//     PlcTask Outputs/GVL_iXlinker.EtherCAT_Master_BKCUCX.TcTerminals210_EK1100_1.TcTerminals210_1BK1250.A_0361_KL_3361_1005_1_Ch_Oscilloscope.Channel_1.Data_Out_8 <-> Channel 1/Data Out 8
//     PlcTask Outputs/GVL_iXlinker.EtherCAT_Master_BKCUCX.TcTerminals210_EK1100_1.TcTerminals210_1BK1250.A_0361_KL_3361_1005_1_Ch_Oscilloscope.Channel_1.Data_Out_9 <-> Channel 1/Data Out 9
//     PlcTask Outputs/GVL_iXlinker.EtherCAT_Master_BKCUCX.TcTerminals210_EK1100_1.TcTerminals210_1BK1250.A_0361_KL_3361_1005_1_Ch_Oscilloscope.Channel_1.Data_Out_10 <-> Channel 1/Data Out 10
//   PLC/PLC Instance <-> EtherCAT Master BKCUCX/TcTerminals210_EK1100_1/TcTerminals210_1BK1250/A_0362(KL 3362, 2 Ch. Oscilloscope)
//     PlcTask Inputs/GVL_iXlinker.EtherCAT_Master_BKCUCX.TcTerminals210_EK1100_1.TcTerminals210_1BK1250.A_0362_KL_3362_2_Ch_Oscilloscope.Channel_1.State <-> Channel 1/State
//     PlcTask Inputs/GVL_iXlinker.EtherCAT_Master_BKCUCX.TcTerminals210_EK1100_1.TcTerminals210_1BK1250.A_0362_KL_3362_2_Ch_Oscilloscope.Channel_2.State <-> Channel 2/State
//     PlcTask Inputs/GVL_iXlinker.EtherCAT_Master_BKCUCX.TcTerminals210_EK1100_1.TcTerminals210_1BK1250.A_0362_KL_3362_2_Ch_Oscilloscope.Channel_1.Data_In <-> Channel 1/Data In
//     PlcTask Inputs/GVL_iXlinker.EtherCAT_Master_BKCUCX.TcTerminals210_EK1100_1.TcTerminals210_1BK1250.A_0362_KL_3362_2_Ch_Oscilloscope.Channel_2.Data_In <-> Channel 2/Data In
//     PlcTask Outputs/GVL_iXlinker.EtherCAT_Master_BKCUCX.TcTerminals210_EK1100_1.TcTerminals210_1BK1250.A_0362_KL_3362_2_Ch_Oscilloscope.Channel_1.Ctrl <-> Channel 1/Ctrl
//     PlcTask Outputs/GVL_iXlinker.EtherCAT_Master_BKCUCX.TcTerminals210_EK1100_1.TcTerminals210_1BK1250.A_0362_KL_3362_2_Ch_Oscilloscope.Channel_2.Ctrl <-> Channel 2/Ctrl
//     PlcTask Outputs/GVL_iXlinker.EtherCAT_Master_BKCUCX.TcTerminals210_EK1100_1.TcTerminals210_1BK1250.A_0362_KL_3362_2_Ch_Oscilloscope.Channel_1.Data_Out <-> Channel 1/Data Out
//     PlcTask Outputs/GVL_iXlinker.EtherCAT_Master_BKCUCX.TcTerminals210_EK1100_1.TcTerminals210_1BK1250.A_0362_KL_3362_2_Ch_Oscilloscope.Channel_2.Data_Out <-> Channel 2/Data Out
//   PLC/PLC Instance <-> EtherCAT Master BKCUCX/TcTerminals210_EK1100_2
//     PlcTask Inputs/GVL_iXlinker.EtherCAT_Master_BKCUCX.TcTerminals210_EK1100_2.InfoData.State <-> InfoData/State
//   PLC/PLC Instance <-> EtherCAT Master BKCUCX/TcTerminals210_EK1100_2/TcTerminals210_2BK1250
//     PlcTask Inputs/GVL_iXlinker.EtherCAT_Master_BKCUCX.TcTerminals210_EK1100_2.TcTerminals210_2BK1250.Inputs.CouplerState <-> Inputs/CouplerState
//     PlcTask Inputs/GVL_iXlinker.EtherCAT_Master_BKCUCX.TcTerminals210_EK1100_2.TcTerminals210_2BK1250.Outputs.CouplerCtrl <-> Outputs/CouplerCtrl
//     PlcTask Inputs/GVL_iXlinker.EtherCAT_Master_BKCUCX.TcTerminals210_EK1100_2.TcTerminals210_2BK1250.WcState.WcState <-> WcState/WcState
//     PlcTask Inputs/GVL_iXlinker.EtherCAT_Master_BKCUCX.TcTerminals210_EK1100_2.TcTerminals210_2BK1250.WcState.InputToggle <-> WcState/InputToggle
//     PlcTask Inputs/GVL_iXlinker.EtherCAT_Master_BKCUCX.TcTerminals210_EK1100_2.TcTerminals210_2BK1250.InfoData.AdsAddr <-> InfoData/AdsAddr
//     PlcTask Inputs/GVL_iXlinker.EtherCAT_Master_BKCUCX.TcTerminals210_EK1100_2.TcTerminals210_2BK1250.InfoData.AoeNetId <-> InfoData/AoeNetId
//     PlcTask Inputs/GVL_iXlinker.EtherCAT_Master_BKCUCX.TcTerminals210_EK1100_2.TcTerminals210_2BK1250.InfoData.State <-> InfoData/State
//   PLC/PLC Instance <-> EtherCAT Master BKCUCX/TcTerminals210_EK1100_2/TcTerminals210_2BK1250/A_0001(KL 6211 ASI-Master (Parameter Interface and 6 Byte (11 ASI-Slaves), Power))
//     PlcTask Inputs/GVL_iXlinker.EtherCAT_Master_BKCUCX.TcTerminals210_EK1100_2.TcTerminals210_2BK1250.A_0001_KL_6211_ASI_Master_Parameter_Interface_and_6_Byte_11_ASI_Slaves_Power.Channel_1.Status <-> Channel 1/Status
//     PlcTask Inputs/GVL_iXlinker.EtherCAT_Master_BKCUCX.TcTerminals210_EK1100_2.TcTerminals210_2BK1250.A_0001_KL_6211_ASI_Master_Parameter_Interface_and_6_Byte_11_ASI_Slaves_Power.Channel_1.Parameter_In <-> Channel 1/Parameter In
//     PlcTask Inputs/GVL_iXlinker.EtherCAT_Master_BKCUCX.TcTerminals210_EK1100_2.TcTerminals210_2BK1250.A_0001_KL_6211_ASI_Master_Parameter_Interface_and_6_Byte_11_ASI_Slaves_Power.Channel_1.ASI_In_Slave_1_Status <-> Channel 1/ASI In Slave 1 Status
//     PlcTask Inputs/GVL_iXlinker.EtherCAT_Master_BKCUCX.TcTerminals210_EK1100_2.TcTerminals210_2BK1250.A_0001_KL_6211_ASI_Master_Parameter_Interface_and_6_Byte_11_ASI_Slaves_Power.Channel_1.ASI_In_Slave_3_Slave_2 <-> Channel 1/ASI In Slave 3 Slave 2
//     PlcTask Inputs/GVL_iXlinker.EtherCAT_Master_BKCUCX.TcTerminals210_EK1100_2.TcTerminals210_2BK1250.A_0001_KL_6211_ASI_Master_Parameter_Interface_and_6_Byte_11_ASI_Slaves_Power.Channel_1.ASI_In_Slave_5_Slave_4 <-> Channel 1/ASI In Slave 5 Slave 4
//     PlcTask Inputs/GVL_iXlinker.EtherCAT_Master_BKCUCX.TcTerminals210_EK1100_2.TcTerminals210_2BK1250.A_0001_KL_6211_ASI_Master_Parameter_Interface_and_6_Byte_11_ASI_Slaves_Power.Channel_1.ASI_In_Slave_7_Slave_6 <-> Channel 1/ASI In Slave 7 Slave 6
//     PlcTask Inputs/GVL_iXlinker.EtherCAT_Master_BKCUCX.TcTerminals210_EK1100_2.TcTerminals210_2BK1250.A_0001_KL_6211_ASI_Master_Parameter_Interface_and_6_Byte_11_ASI_Slaves_Power.Channel_1.ASI_In_Slave_9_Slave_8 <-> Channel 1/ASI In Slave 9 Slave 8
//     PlcTask Inputs/GVL_iXlinker.EtherCAT_Master_BKCUCX.TcTerminals210_EK1100_2.TcTerminals210_2BK1250.A_0001_KL_6211_ASI_Master_Parameter_Interface_and_6_Byte_11_ASI_Slaves_Power.Channel_1.ASI_In_Slave_11_Slave_10 <-> Channel 1/ASI In Slave 11 Slave 10
//     PlcTask Outputs/GVL_iXlinker.EtherCAT_Master_BKCUCX.TcTerminals210_EK1100_2.TcTerminals210_2BK1250.A_0001_KL_6211_ASI_Master_Parameter_Interface_and_6_Byte_11_ASI_Slaves_Power.Channel_1.Control <-> Channel 1/Control
//     PlcTask Outputs/GVL_iXlinker.EtherCAT_Master_BKCUCX.TcTerminals210_EK1100_2.TcTerminals210_2BK1250.A_0001_KL_6211_ASI_Master_Parameter_Interface_and_6_Byte_11_ASI_Slaves_Power.Channel_1.Parameter_Out <-> Channel 1/Parameter Out
//     PlcTask Outputs/GVL_iXlinker.EtherCAT_Master_BKCUCX.TcTerminals210_EK1100_2.TcTerminals210_2BK1250.A_0001_KL_6211_ASI_Master_Parameter_Interface_and_6_Byte_11_ASI_Slaves_Power.Channel_1.ASI_Out_Slave_1_Control <-> Channel 1/ASI Out Slave 1 Control
//     PlcTask Outputs/GVL_iXlinker.EtherCAT_Master_BKCUCX.TcTerminals210_EK1100_2.TcTerminals210_2BK1250.A_0001_KL_6211_ASI_Master_Parameter_Interface_and_6_Byte_11_ASI_Slaves_Power.Channel_1.ASI_Out_Slave_3_Slave_2 <-> Channel 1/ASI Out Slave 3 Slave 2
//     PlcTask Outputs/GVL_iXlinker.EtherCAT_Master_BKCUCX.TcTerminals210_EK1100_2.TcTerminals210_2BK1250.A_0001_KL_6211_ASI_Master_Parameter_Interface_and_6_Byte_11_ASI_Slaves_Power.Channel_1.ASI_Out_Slave_5_Slave_4 <-> Channel 1/ASI Out Slave 5 Slave 4
//     PlcTask Outputs/GVL_iXlinker.EtherCAT_Master_BKCUCX.TcTerminals210_EK1100_2.TcTerminals210_2BK1250.A_0001_KL_6211_ASI_Master_Parameter_Interface_and_6_Byte_11_ASI_Slaves_Power.Channel_1.ASI_Out_Slave_7_Slave_6 <-> Channel 1/ASI Out Slave 7 Slave 6
//     PlcTask Outputs/GVL_iXlinker.EtherCAT_Master_BKCUCX.TcTerminals210_EK1100_2.TcTerminals210_2BK1250.A_0001_KL_6211_ASI_Master_Parameter_Interface_and_6_Byte_11_ASI_Slaves_Power.Channel_1.ASI_Out_Slave_9_Slave_8 <-> Channel 1/ASI Out Slave 9 Slave 8
//     PlcTask Outputs/GVL_iXlinker.EtherCAT_Master_BKCUCX.TcTerminals210_EK1100_2.TcTerminals210_2BK1250.A_0001_KL_6211_ASI_Master_Parameter_Interface_and_6_Byte_11_ASI_Slaves_Power.Channel_1.ASI_Out_Slave_11_Slave_10 <-> Channel 1/ASI Out Slave 11 Slave 10
//   PLC/PLC Instance <-> EtherCAT Master BKCUCX/TcTerminals210_EK1100_2/TcTerminals210_2BK1250/A_0002(KL 6211 ASI-Master (Parameter Interface and 6 Byte (11 ASI-Slaves), Power))
//     PlcTask Inputs/GVL_iXlinker.EtherCAT_Master_BKCUCX.TcTerminals210_EK1100_2.TcTerminals210_2BK1250.A_0002_KL_6211_ASI_Master_Parameter_Interface_and_6_Byte_11_ASI_Slaves_Power.Channel_1.Status <-> Channel 1/Status
//     PlcTask Inputs/GVL_iXlinker.EtherCAT_Master_BKCUCX.TcTerminals210_EK1100_2.TcTerminals210_2BK1250.A_0002_KL_6211_ASI_Master_Parameter_Interface_and_6_Byte_11_ASI_Slaves_Power.Channel_1.Parameter_In <-> Channel 1/Parameter In
//     PlcTask Inputs/GVL_iXlinker.EtherCAT_Master_BKCUCX.TcTerminals210_EK1100_2.TcTerminals210_2BK1250.A_0002_KL_6211_ASI_Master_Parameter_Interface_and_6_Byte_11_ASI_Slaves_Power.Channel_1.ASI_In_Status <-> Channel 1/ASI In Status
//     PlcTask Inputs/GVL_iXlinker.EtherCAT_Master_BKCUCX.TcTerminals210_EK1100_2.TcTerminals210_2BK1250.A_0002_KL_6211_ASI_Master_Parameter_Interface_and_6_Byte_11_ASI_Slaves_Power.Channel_1.ASI_In_Slave_1 <-> Channel 1/ASI In Slave 1
//     PlcTask Inputs/GVL_iXlinker.EtherCAT_Master_BKCUCX.TcTerminals210_EK1100_2.TcTerminals210_2BK1250.A_0002_KL_6211_ASI_Master_Parameter_Interface_and_6_Byte_11_ASI_Slaves_Power.Channel_1.ASI_In_Slave_2 <-> Channel 1/ASI In Slave 2
//     PlcTask Inputs/GVL_iXlinker.EtherCAT_Master_BKCUCX.TcTerminals210_EK1100_2.TcTerminals210_2BK1250.A_0002_KL_6211_ASI_Master_Parameter_Interface_and_6_Byte_11_ASI_Slaves_Power.Channel_1.ASI_In_Slave_3 <-> Channel 1/ASI In Slave 3
//     PlcTask Inputs/GVL_iXlinker.EtherCAT_Master_BKCUCX.TcTerminals210_EK1100_2.TcTerminals210_2BK1250.A_0002_KL_6211_ASI_Master_Parameter_Interface_and_6_Byte_11_ASI_Slaves_Power.Channel_1.ASI_In_Slave_4 <-> Channel 1/ASI In Slave 4
//     PlcTask Inputs/GVL_iXlinker.EtherCAT_Master_BKCUCX.TcTerminals210_EK1100_2.TcTerminals210_2BK1250.A_0002_KL_6211_ASI_Master_Parameter_Interface_and_6_Byte_11_ASI_Slaves_Power.Channel_1.ASI_In_Slave_5 <-> Channel 1/ASI In Slave 5
//     PlcTask Inputs/GVL_iXlinker.EtherCAT_Master_BKCUCX.TcTerminals210_EK1100_2.TcTerminals210_2BK1250.A_0002_KL_6211_ASI_Master_Parameter_Interface_and_6_Byte_11_ASI_Slaves_Power.Channel_1.ASI_In_Slave_6 <-> Channel 1/ASI In Slave 6
//     PlcTask Inputs/GVL_iXlinker.EtherCAT_Master_BKCUCX.TcTerminals210_EK1100_2.TcTerminals210_2BK1250.A_0002_KL_6211_ASI_Master_Parameter_Interface_and_6_Byte_11_ASI_Slaves_Power.Channel_1.ASI_In_Slave_7 <-> Channel 1/ASI In Slave 7
//     PlcTask Inputs/GVL_iXlinker.EtherCAT_Master_BKCUCX.TcTerminals210_EK1100_2.TcTerminals210_2BK1250.A_0002_KL_6211_ASI_Master_Parameter_Interface_and_6_Byte_11_ASI_Slaves_Power.Channel_1.ASI_In_Slave_8 <-> Channel 1/ASI In Slave 8
//     PlcTask Inputs/GVL_iXlinker.EtherCAT_Master_BKCUCX.TcTerminals210_EK1100_2.TcTerminals210_2BK1250.A_0002_KL_6211_ASI_Master_Parameter_Interface_and_6_Byte_11_ASI_Slaves_Power.Channel_1.ASI_In_Slave_9 <-> Channel 1/ASI In Slave 9
//     PlcTask Inputs/GVL_iXlinker.EtherCAT_Master_BKCUCX.TcTerminals210_EK1100_2.TcTerminals210_2BK1250.A_0002_KL_6211_ASI_Master_Parameter_Interface_and_6_Byte_11_ASI_Slaves_Power.Channel_1.ASI_In_Slave_10 <-> Channel 1/ASI In Slave 10
//     PlcTask Inputs/GVL_iXlinker.EtherCAT_Master_BKCUCX.TcTerminals210_EK1100_2.TcTerminals210_2BK1250.A_0002_KL_6211_ASI_Master_Parameter_Interface_and_6_Byte_11_ASI_Slaves_Power.Channel_1.ASI_In_Slave_11 <-> Channel 1/ASI In Slave 11
//     PlcTask Outputs/GVL_iXlinker.EtherCAT_Master_BKCUCX.TcTerminals210_EK1100_2.TcTerminals210_2BK1250.A_0002_KL_6211_ASI_Master_Parameter_Interface_and_6_Byte_11_ASI_Slaves_Power.Channel_1.Control <-> Channel 1/Control
//     PlcTask Outputs/GVL_iXlinker.EtherCAT_Master_BKCUCX.TcTerminals210_EK1100_2.TcTerminals210_2BK1250.A_0002_KL_6211_ASI_Master_Parameter_Interface_and_6_Byte_11_ASI_Slaves_Power.Channel_1.Parameter_Out <-> Channel 1/Parameter Out
//     PlcTask Outputs/GVL_iXlinker.EtherCAT_Master_BKCUCX.TcTerminals210_EK1100_2.TcTerminals210_2BK1250.A_0002_KL_6211_ASI_Master_Parameter_Interface_and_6_Byte_11_ASI_Slaves_Power.Channel_1.ASI_Out_Control <-> Channel 1/ASI Out Control
//     PlcTask Outputs/GVL_iXlinker.EtherCAT_Master_BKCUCX.TcTerminals210_EK1100_2.TcTerminals210_2BK1250.A_0002_KL_6211_ASI_Master_Parameter_Interface_and_6_Byte_11_ASI_Slaves_Power.Channel_1.ASI_Out_Slave_1 <-> Channel 1/ASI Out Slave 1
//     PlcTask Outputs/GVL_iXlinker.EtherCAT_Master_BKCUCX.TcTerminals210_EK1100_2.TcTerminals210_2BK1250.A_0002_KL_6211_ASI_Master_Parameter_Interface_and_6_Byte_11_ASI_Slaves_Power.Channel_1.ASI_Out_Slave_2 <-> Channel 1/ASI Out Slave 2
//     PlcTask Outputs/GVL_iXlinker.EtherCAT_Master_BKCUCX.TcTerminals210_EK1100_2.TcTerminals210_2BK1250.A_0002_KL_6211_ASI_Master_Parameter_Interface_and_6_Byte_11_ASI_Slaves_Power.Channel_1.ASI_Out_Slave_3 <-> Channel 1/ASI Out Slave 3
//     PlcTask Outputs/GVL_iXlinker.EtherCAT_Master_BKCUCX.TcTerminals210_EK1100_2.TcTerminals210_2BK1250.A_0002_KL_6211_ASI_Master_Parameter_Interface_and_6_Byte_11_ASI_Slaves_Power.Channel_1.ASI_Out_Slave_4 <-> Channel 1/ASI Out Slave 4
//     PlcTask Outputs/GVL_iXlinker.EtherCAT_Master_BKCUCX.TcTerminals210_EK1100_2.TcTerminals210_2BK1250.A_0002_KL_6211_ASI_Master_Parameter_Interface_and_6_Byte_11_ASI_Slaves_Power.Channel_1.ASI_Out_Slave_5 <-> Channel 1/ASI Out Slave 5
//     PlcTask Outputs/GVL_iXlinker.EtherCAT_Master_BKCUCX.TcTerminals210_EK1100_2.TcTerminals210_2BK1250.A_0002_KL_6211_ASI_Master_Parameter_Interface_and_6_Byte_11_ASI_Slaves_Power.Channel_1.ASI_Out_Slave_6 <-> Channel 1/ASI Out Slave 6
//     PlcTask Outputs/GVL_iXlinker.EtherCAT_Master_BKCUCX.TcTerminals210_EK1100_2.TcTerminals210_2BK1250.A_0002_KL_6211_ASI_Master_Parameter_Interface_and_6_Byte_11_ASI_Slaves_Power.Channel_1.ASI_Out_Slave_7 <-> Channel 1/ASI Out Slave 7
//     PlcTask Outputs/GVL_iXlinker.EtherCAT_Master_BKCUCX.TcTerminals210_EK1100_2.TcTerminals210_2BK1250.A_0002_KL_6211_ASI_Master_Parameter_Interface_and_6_Byte_11_ASI_Slaves_Power.Channel_1.ASI_Out_Slave_8 <-> Channel 1/ASI Out Slave 8
//     PlcTask Outputs/GVL_iXlinker.EtherCAT_Master_BKCUCX.TcTerminals210_EK1100_2.TcTerminals210_2BK1250.A_0002_KL_6211_ASI_Master_Parameter_Interface_and_6_Byte_11_ASI_Slaves_Power.Channel_1.ASI_Out_Slave_9 <-> Channel 1/ASI Out Slave 9
//     PlcTask Outputs/GVL_iXlinker.EtherCAT_Master_BKCUCX.TcTerminals210_EK1100_2.TcTerminals210_2BK1250.A_0002_KL_6211_ASI_Master_Parameter_Interface_and_6_Byte_11_ASI_Slaves_Power.Channel_1.ASI_Out_Slave_10 <-> Channel 1/ASI Out Slave 10
//     PlcTask Outputs/GVL_iXlinker.EtherCAT_Master_BKCUCX.TcTerminals210_EK1100_2.TcTerminals210_2BK1250.A_0002_KL_6211_ASI_Master_Parameter_Interface_and_6_Byte_11_ASI_Slaves_Power.Channel_1.ASI_Out_Slave_11 <-> Channel 1/ASI Out Slave 11
//   PLC/PLC Instance <-> EtherCAT Master BKCUCX/TcTerminals210_EK1100_2/TcTerminals210_2BK1250/A_0005(KL 6211 ASI-Master (Parameter Interface and 16 Byte (31 ASI-Slaves), Power))
//     PlcTask Inputs/GVL_iXlinker.EtherCAT_Master_BKCUCX.TcTerminals210_EK1100_2.TcTerminals210_2BK1250.A_0005_KL_6211_ASI_Master_Parameter_Interface_and_16_Byte_31_ASI_Slaves_Power.Channel_1.Status <-> Channel 1/Status
//     PlcTask Inputs/GVL_iXlinker.EtherCAT_Master_BKCUCX.TcTerminals210_EK1100_2.TcTerminals210_2BK1250.A_0005_KL_6211_ASI_Master_Parameter_Interface_and_16_Byte_31_ASI_Slaves_Power.Channel_1.Parameter_In <-> Channel 1/Parameter In
//     PlcTask Inputs/GVL_iXlinker.EtherCAT_Master_BKCUCX.TcTerminals210_EK1100_2.TcTerminals210_2BK1250.A_0005_KL_6211_ASI_Master_Parameter_Interface_and_16_Byte_31_ASI_Slaves_Power.Channel_1.ASI_In_Slave_1_Status <-> Channel 1/ASI In Slave 1 Status
//     PlcTask Inputs/GVL_iXlinker.EtherCAT_Master_BKCUCX.TcTerminals210_EK1100_2.TcTerminals210_2BK1250.A_0005_KL_6211_ASI_Master_Parameter_Interface_and_16_Byte_31_ASI_Slaves_Power.Channel_1.ASI_In_Slave_3_Slave_2 <-> Channel 1/ASI In Slave 3 Slave 2
//     PlcTask Inputs/GVL_iXlinker.EtherCAT_Master_BKCUCX.TcTerminals210_EK1100_2.TcTerminals210_2BK1250.A_0005_KL_6211_ASI_Master_Parameter_Interface_and_16_Byte_31_ASI_Slaves_Power.Channel_1.ASI_In_Slave_5_Slave_4 <-> Channel 1/ASI In Slave 5 Slave 4
//     PlcTask Inputs/GVL_iXlinker.EtherCAT_Master_BKCUCX.TcTerminals210_EK1100_2.TcTerminals210_2BK1250.A_0005_KL_6211_ASI_Master_Parameter_Interface_and_16_Byte_31_ASI_Slaves_Power.Channel_1.ASI_In_Slave_7_Slave_6 <-> Channel 1/ASI In Slave 7 Slave 6
//     PlcTask Inputs/GVL_iXlinker.EtherCAT_Master_BKCUCX.TcTerminals210_EK1100_2.TcTerminals210_2BK1250.A_0005_KL_6211_ASI_Master_Parameter_Interface_and_16_Byte_31_ASI_Slaves_Power.Channel_1.ASI_In_Slave_9_Slave_8 <-> Channel 1/ASI In Slave 9 Slave 8
//     PlcTask Inputs/GVL_iXlinker.EtherCAT_Master_BKCUCX.TcTerminals210_EK1100_2.TcTerminals210_2BK1250.A_0005_KL_6211_ASI_Master_Parameter_Interface_and_16_Byte_31_ASI_Slaves_Power.Channel_1.ASI_In_Slave_11_Slave_10 <-> Channel 1/ASI In Slave 11 Slave 10
//     PlcTask Inputs/GVL_iXlinker.EtherCAT_Master_BKCUCX.TcTerminals210_EK1100_2.TcTerminals210_2BK1250.A_0005_KL_6211_ASI_Master_Parameter_Interface_and_16_Byte_31_ASI_Slaves_Power.Channel_1.ASI_In_Slave_13_Slave_12 <-> Channel 1/ASI In Slave 13 Slave 12
//     PlcTask Inputs/GVL_iXlinker.EtherCAT_Master_BKCUCX.TcTerminals210_EK1100_2.TcTerminals210_2BK1250.A_0005_KL_6211_ASI_Master_Parameter_Interface_and_16_Byte_31_ASI_Slaves_Power.Channel_1.ASI_In_Slave_15_Slave_14 <-> Channel 1/ASI In Slave 15 Slave 14
//     PlcTask Inputs/GVL_iXlinker.EtherCAT_Master_BKCUCX.TcTerminals210_EK1100_2.TcTerminals210_2BK1250.A_0005_KL_6211_ASI_Master_Parameter_Interface_and_16_Byte_31_ASI_Slaves_Power.Channel_1.ASI_In_Slave_17_Slave_16 <-> Channel 1/ASI In Slave 17 Slave 16
//     PlcTask Inputs/GVL_iXlinker.EtherCAT_Master_BKCUCX.TcTerminals210_EK1100_2.TcTerminals210_2BK1250.A_0005_KL_6211_ASI_Master_Parameter_Interface_and_16_Byte_31_ASI_Slaves_Power.Channel_1.ASI_In_Slave_19_Slave_18 <-> Channel 1/ASI In Slave 19 Slave 18
//     PlcTask Inputs/GVL_iXlinker.EtherCAT_Master_BKCUCX.TcTerminals210_EK1100_2.TcTerminals210_2BK1250.A_0005_KL_6211_ASI_Master_Parameter_Interface_and_16_Byte_31_ASI_Slaves_Power.Channel_1.ASI_In_Slave_21_Slave_20 <-> Channel 1/ASI In Slave 21 Slave 20
//     PlcTask Inputs/GVL_iXlinker.EtherCAT_Master_BKCUCX.TcTerminals210_EK1100_2.TcTerminals210_2BK1250.A_0005_KL_6211_ASI_Master_Parameter_Interface_and_16_Byte_31_ASI_Slaves_Power.Channel_1.ASI_In_Slave_23_Slave_22 <-> Channel 1/ASI In Slave 23 Slave 22
//     PlcTask Inputs/GVL_iXlinker.EtherCAT_Master_BKCUCX.TcTerminals210_EK1100_2.TcTerminals210_2BK1250.A_0005_KL_6211_ASI_Master_Parameter_Interface_and_16_Byte_31_ASI_Slaves_Power.Channel_1.ASI_In_Slave_25_Slave_24 <-> Channel 1/ASI In Slave 25 Slave 24
//     PlcTask Inputs/GVL_iXlinker.EtherCAT_Master_BKCUCX.TcTerminals210_EK1100_2.TcTerminals210_2BK1250.A_0005_KL_6211_ASI_Master_Parameter_Interface_and_16_Byte_31_ASI_Slaves_Power.Channel_1.ASI_In_Slave_27_Slave_26 <-> Channel 1/ASI In Slave 27 Slave 26
//     PlcTask Inputs/GVL_iXlinker.EtherCAT_Master_BKCUCX.TcTerminals210_EK1100_2.TcTerminals210_2BK1250.A_0005_KL_6211_ASI_Master_Parameter_Interface_and_16_Byte_31_ASI_Slaves_Power.Channel_1.ASI_In_Slave_29_Slave_28 <-> Channel 1/ASI In Slave 29 Slave 28
//     PlcTask Inputs/GVL_iXlinker.EtherCAT_Master_BKCUCX.TcTerminals210_EK1100_2.TcTerminals210_2BK1250.A_0005_KL_6211_ASI_Master_Parameter_Interface_and_16_Byte_31_ASI_Slaves_Power.Channel_1.ASI_In_Slave_31_Slave_30 <-> Channel 1/ASI In Slave 31 Slave 30
//     PlcTask Outputs/GVL_iXlinker.EtherCAT_Master_BKCUCX.TcTerminals210_EK1100_2.TcTerminals210_2BK1250.A_0005_KL_6211_ASI_Master_Parameter_Interface_and_16_Byte_31_ASI_Slaves_Power.Channel_1.Control <-> Channel 1/Control
//     PlcTask Outputs/GVL_iXlinker.EtherCAT_Master_BKCUCX.TcTerminals210_EK1100_2.TcTerminals210_2BK1250.A_0005_KL_6211_ASI_Master_Parameter_Interface_and_16_Byte_31_ASI_Slaves_Power.Channel_1.Parameter_Out <-> Channel 1/Parameter Out
//     PlcTask Outputs/GVL_iXlinker.EtherCAT_Master_BKCUCX.TcTerminals210_EK1100_2.TcTerminals210_2BK1250.A_0005_KL_6211_ASI_Master_Parameter_Interface_and_16_Byte_31_ASI_Slaves_Power.Channel_1.ASI_Out_Slave_1_Control <-> Channel 1/ASI Out Slave 1 Control
//     PlcTask Outputs/GVL_iXlinker.EtherCAT_Master_BKCUCX.TcTerminals210_EK1100_2.TcTerminals210_2BK1250.A_0005_KL_6211_ASI_Master_Parameter_Interface_and_16_Byte_31_ASI_Slaves_Power.Channel_1.ASI_Out_Slave_3_Slave_2 <-> Channel 1/ASI Out Slave 3 Slave 2
//     PlcTask Outputs/GVL_iXlinker.EtherCAT_Master_BKCUCX.TcTerminals210_EK1100_2.TcTerminals210_2BK1250.A_0005_KL_6211_ASI_Master_Parameter_Interface_and_16_Byte_31_ASI_Slaves_Power.Channel_1.ASI_Out_Slave_5_Slave_4 <-> Channel 1/ASI Out Slave 5 Slave 4
//     PlcTask Outputs/GVL_iXlinker.EtherCAT_Master_BKCUCX.TcTerminals210_EK1100_2.TcTerminals210_2BK1250.A_0005_KL_6211_ASI_Master_Parameter_Interface_and_16_Byte_31_ASI_Slaves_Power.Channel_1.ASI_Out_Slave_7_Slave_6 <-> Channel 1/ASI Out Slave 7 Slave 6
//     PlcTask Outputs/GVL_iXlinker.EtherCAT_Master_BKCUCX.TcTerminals210_EK1100_2.TcTerminals210_2BK1250.A_0005_KL_6211_ASI_Master_Parameter_Interface_and_16_Byte_31_ASI_Slaves_Power.Channel_1.ASI_Out_Slave_9_Slave_8 <-> Channel 1/ASI Out Slave 9 Slave 8
//     PlcTask Outputs/GVL_iXlinker.EtherCAT_Master_BKCUCX.TcTerminals210_EK1100_2.TcTerminals210_2BK1250.A_0005_KL_6211_ASI_Master_Parameter_Interface_and_16_Byte_31_ASI_Slaves_Power.Channel_1.ASI_Out_Slave_11_Slave_10 <-> Channel 1/ASI Out Slave 11 Slave 10
//     PlcTask Outputs/GVL_iXlinker.EtherCAT_Master_BKCUCX.TcTerminals210_EK1100_2.TcTerminals210_2BK1250.A_0005_KL_6211_ASI_Master_Parameter_Interface_and_16_Byte_31_ASI_Slaves_Power.Channel_1.ASI_Out_Slave_13_Slave_12 <-> Channel 1/ASI Out Slave 13 Slave 12
//     PlcTask Outputs/GVL_iXlinker.EtherCAT_Master_BKCUCX.TcTerminals210_EK1100_2.TcTerminals210_2BK1250.A_0005_KL_6211_ASI_Master_Parameter_Interface_and_16_Byte_31_ASI_Slaves_Power.Channel_1.ASI_Out_Slave_15_Slave_14 <-> Channel 1/ASI Out Slave 15 Slave 14
//     PlcTask Outputs/GVL_iXlinker.EtherCAT_Master_BKCUCX.TcTerminals210_EK1100_2.TcTerminals210_2BK1250.A_0005_KL_6211_ASI_Master_Parameter_Interface_and_16_Byte_31_ASI_Slaves_Power.Channel_1.ASI_Out_Slave_17_Slave_16 <-> Channel 1/ASI Out Slave 17 Slave 16
//     PlcTask Outputs/GVL_iXlinker.EtherCAT_Master_BKCUCX.TcTerminals210_EK1100_2.TcTerminals210_2BK1250.A_0005_KL_6211_ASI_Master_Parameter_Interface_and_16_Byte_31_ASI_Slaves_Power.Channel_1.ASI_Out_Slave_19_Slave_18 <-> Channel 1/ASI Out Slave 19 Slave 18
//     PlcTask Outputs/GVL_iXlinker.EtherCAT_Master_BKCUCX.TcTerminals210_EK1100_2.TcTerminals210_2BK1250.A_0005_KL_6211_ASI_Master_Parameter_Interface_and_16_Byte_31_ASI_Slaves_Power.Channel_1.ASI_Out_Slave_21_Slave_20 <-> Channel 1/ASI Out Slave 21 Slave 20
//     PlcTask Outputs/GVL_iXlinker.EtherCAT_Master_BKCUCX.TcTerminals210_EK1100_2.TcTerminals210_2BK1250.A_0005_KL_6211_ASI_Master_Parameter_Interface_and_16_Byte_31_ASI_Slaves_Power.Channel_1.ASI_Out_Slave_23_Slave_22 <-> Channel 1/ASI Out Slave 23 Slave 22
//     PlcTask Outputs/GVL_iXlinker.EtherCAT_Master_BKCUCX.TcTerminals210_EK1100_2.TcTerminals210_2BK1250.A_0005_KL_6211_ASI_Master_Parameter_Interface_and_16_Byte_31_ASI_Slaves_Power.Channel_1.ASI_Out_Slave_25_Slave_24 <-> Channel 1/ASI Out Slave 25 Slave 24
//     PlcTask Outputs/GVL_iXlinker.EtherCAT_Master_BKCUCX.TcTerminals210_EK1100_2.TcTerminals210_2BK1250.A_0005_KL_6211_ASI_Master_Parameter_Interface_and_16_Byte_31_ASI_Slaves_Power.Channel_1.ASI_Out_Slave_27_Slave_26 <-> Channel 1/ASI Out Slave 27 Slave 26
//     PlcTask Outputs/GVL_iXlinker.EtherCAT_Master_BKCUCX.TcTerminals210_EK1100_2.TcTerminals210_2BK1250.A_0005_KL_6211_ASI_Master_Parameter_Interface_and_16_Byte_31_ASI_Slaves_Power.Channel_1.ASI_Out_Slave_29_Slave_28 <-> Channel 1/ASI Out Slave 29 Slave 28
//     PlcTask Outputs/GVL_iXlinker.EtherCAT_Master_BKCUCX.TcTerminals210_EK1100_2.TcTerminals210_2BK1250.A_0005_KL_6211_ASI_Master_Parameter_Interface_and_16_Byte_31_ASI_Slaves_Power.Channel_1.ASI_Out_Slave_31_Slave_30 <-> Channel 1/ASI Out Slave 31 Slave 30
//   PLC/PLC Instance <-> EtherCAT Master BKCUCX/TcTerminals210_EK1100_2/TcTerminals210_2BK1250/A_0006(KL 6211 ASI-Master (Parameter Interface and 16 Byte (31 ASI-Slaves), Power))
//     PlcTask Inputs/GVL_iXlinker.EtherCAT_Master_BKCUCX.TcTerminals210_EK1100_2.TcTerminals210_2BK1250.A_0006_KL_6211_ASI_Master_Parameter_Interface_and_16_Byte_31_ASI_Slaves_Power.Channel_1.Status <-> Channel 1/Status
//     PlcTask Inputs/GVL_iXlinker.EtherCAT_Master_BKCUCX.TcTerminals210_EK1100_2.TcTerminals210_2BK1250.A_0006_KL_6211_ASI_Master_Parameter_Interface_and_16_Byte_31_ASI_Slaves_Power.Channel_1.Parameter_In <-> Channel 1/Parameter In
//     PlcTask Inputs/GVL_iXlinker.EtherCAT_Master_BKCUCX.TcTerminals210_EK1100_2.TcTerminals210_2BK1250.A_0006_KL_6211_ASI_Master_Parameter_Interface_and_16_Byte_31_ASI_Slaves_Power.Channel_1.ASI_In_Status <-> Channel 1/ASI In Status
//     PlcTask Inputs/GVL_iXlinker.EtherCAT_Master_BKCUCX.TcTerminals210_EK1100_2.TcTerminals210_2BK1250.A_0006_KL_6211_ASI_Master_Parameter_Interface_and_16_Byte_31_ASI_Slaves_Power.Channel_1.ASI_In_Slave_1 <-> Channel 1/ASI In Slave 1
//     PlcTask Inputs/GVL_iXlinker.EtherCAT_Master_BKCUCX.TcTerminals210_EK1100_2.TcTerminals210_2BK1250.A_0006_KL_6211_ASI_Master_Parameter_Interface_and_16_Byte_31_ASI_Slaves_Power.Channel_1.ASI_In_Slave_2 <-> Channel 1/ASI In Slave 2
//     PlcTask Inputs/GVL_iXlinker.EtherCAT_Master_BKCUCX.TcTerminals210_EK1100_2.TcTerminals210_2BK1250.A_0006_KL_6211_ASI_Master_Parameter_Interface_and_16_Byte_31_ASI_Slaves_Power.Channel_1.ASI_In_Slave_3 <-> Channel 1/ASI In Slave 3
//     PlcTask Inputs/GVL_iXlinker.EtherCAT_Master_BKCUCX.TcTerminals210_EK1100_2.TcTerminals210_2BK1250.A_0006_KL_6211_ASI_Master_Parameter_Interface_and_16_Byte_31_ASI_Slaves_Power.Channel_1.ASI_In_Slave_4 <-> Channel 1/ASI In Slave 4
//     PlcTask Inputs/GVL_iXlinker.EtherCAT_Master_BKCUCX.TcTerminals210_EK1100_2.TcTerminals210_2BK1250.A_0006_KL_6211_ASI_Master_Parameter_Interface_and_16_Byte_31_ASI_Slaves_Power.Channel_1.ASI_In_Slave_5 <-> Channel 1/ASI In Slave 5
//     PlcTask Inputs/GVL_iXlinker.EtherCAT_Master_BKCUCX.TcTerminals210_EK1100_2.TcTerminals210_2BK1250.A_0006_KL_6211_ASI_Master_Parameter_Interface_and_16_Byte_31_ASI_Slaves_Power.Channel_1.ASI_In_Slave_6 <-> Channel 1/ASI In Slave 6
//     PlcTask Inputs/GVL_iXlinker.EtherCAT_Master_BKCUCX.TcTerminals210_EK1100_2.TcTerminals210_2BK1250.A_0006_KL_6211_ASI_Master_Parameter_Interface_and_16_Byte_31_ASI_Slaves_Power.Channel_1.ASI_In_Slave_7 <-> Channel 1/ASI In Slave 7
//     PlcTask Inputs/GVL_iXlinker.EtherCAT_Master_BKCUCX.TcTerminals210_EK1100_2.TcTerminals210_2BK1250.A_0006_KL_6211_ASI_Master_Parameter_Interface_and_16_Byte_31_ASI_Slaves_Power.Channel_1.ASI_In_Slave_8 <-> Channel 1/ASI In Slave 8
//     PlcTask Inputs/GVL_iXlinker.EtherCAT_Master_BKCUCX.TcTerminals210_EK1100_2.TcTerminals210_2BK1250.A_0006_KL_6211_ASI_Master_Parameter_Interface_and_16_Byte_31_ASI_Slaves_Power.Channel_1.ASI_In_Slave_9 <-> Channel 1/ASI In Slave 9
//     PlcTask Inputs/GVL_iXlinker.EtherCAT_Master_BKCUCX.TcTerminals210_EK1100_2.TcTerminals210_2BK1250.A_0006_KL_6211_ASI_Master_Parameter_Interface_and_16_Byte_31_ASI_Slaves_Power.Channel_1.ASI_In_Slave_10 <-> Channel 1/ASI In Slave 10
//     PlcTask Inputs/GVL_iXlinker.EtherCAT_Master_BKCUCX.TcTerminals210_EK1100_2.TcTerminals210_2BK1250.A_0006_KL_6211_ASI_Master_Parameter_Interface_and_16_Byte_31_ASI_Slaves_Power.Channel_1.ASI_In_Slave_11 <-> Channel 1/ASI In Slave 11
//     PlcTask Inputs/GVL_iXlinker.EtherCAT_Master_BKCUCX.TcTerminals210_EK1100_2.TcTerminals210_2BK1250.A_0006_KL_6211_ASI_Master_Parameter_Interface_and_16_Byte_31_ASI_Slaves_Power.Channel_1.ASI_In_Slave_12 <-> Channel 1/ASI In Slave 12
//     PlcTask Inputs/GVL_iXlinker.EtherCAT_Master_BKCUCX.TcTerminals210_EK1100_2.TcTerminals210_2BK1250.A_0006_KL_6211_ASI_Master_Parameter_Interface_and_16_Byte_31_ASI_Slaves_Power.Channel_1.ASI_In_Slave_13 <-> Channel 1/ASI In Slave 13
//     PlcTask Inputs/GVL_iXlinker.EtherCAT_Master_BKCUCX.TcTerminals210_EK1100_2.TcTerminals210_2BK1250.A_0006_KL_6211_ASI_Master_Parameter_Interface_and_16_Byte_31_ASI_Slaves_Power.Channel_1.ASI_In_Slave_14 <-> Channel 1/ASI In Slave 14
//     PlcTask Inputs/GVL_iXlinker.EtherCAT_Master_BKCUCX.TcTerminals210_EK1100_2.TcTerminals210_2BK1250.A_0006_KL_6211_ASI_Master_Parameter_Interface_and_16_Byte_31_ASI_Slaves_Power.Channel_1.ASI_In_Slave_15 <-> Channel 1/ASI In Slave 15
//     PlcTask Inputs/GVL_iXlinker.EtherCAT_Master_BKCUCX.TcTerminals210_EK1100_2.TcTerminals210_2BK1250.A_0006_KL_6211_ASI_Master_Parameter_Interface_and_16_Byte_31_ASI_Slaves_Power.Channel_1.ASI_In_Slave_16 <-> Channel 1/ASI In Slave 16
//     PlcTask Inputs/GVL_iXlinker.EtherCAT_Master_BKCUCX.TcTerminals210_EK1100_2.TcTerminals210_2BK1250.A_0006_KL_6211_ASI_Master_Parameter_Interface_and_16_Byte_31_ASI_Slaves_Power.Channel_1.ASI_In_Slave_17 <-> Channel 1/ASI In Slave 17
//     PlcTask Inputs/GVL_iXlinker.EtherCAT_Master_BKCUCX.TcTerminals210_EK1100_2.TcTerminals210_2BK1250.A_0006_KL_6211_ASI_Master_Parameter_Interface_and_16_Byte_31_ASI_Slaves_Power.Channel_1.ASI_In_Slave_18 <-> Channel 1/ASI In Slave 18
//     PlcTask Inputs/GVL_iXlinker.EtherCAT_Master_BKCUCX.TcTerminals210_EK1100_2.TcTerminals210_2BK1250.A_0006_KL_6211_ASI_Master_Parameter_Interface_and_16_Byte_31_ASI_Slaves_Power.Channel_1.ASI_In_Slave_19 <-> Channel 1/ASI In Slave 19
//     PlcTask Inputs/GVL_iXlinker.EtherCAT_Master_BKCUCX.TcTerminals210_EK1100_2.TcTerminals210_2BK1250.A_0006_KL_6211_ASI_Master_Parameter_Interface_and_16_Byte_31_ASI_Slaves_Power.Channel_1.ASI_In_Slave_20 <-> Channel 1/ASI In Slave 20
//     PlcTask Inputs/GVL_iXlinker.EtherCAT_Master_BKCUCX.TcTerminals210_EK1100_2.TcTerminals210_2BK1250.A_0006_KL_6211_ASI_Master_Parameter_Interface_and_16_Byte_31_ASI_Slaves_Power.Channel_1.ASI_In_Slave_21 <-> Channel 1/ASI In Slave 21
//     PlcTask Inputs/GVL_iXlinker.EtherCAT_Master_BKCUCX.TcTerminals210_EK1100_2.TcTerminals210_2BK1250.A_0006_KL_6211_ASI_Master_Parameter_Interface_and_16_Byte_31_ASI_Slaves_Power.Channel_1.ASI_In_Slave_22 <-> Channel 1/ASI In Slave 22
//     PlcTask Inputs/GVL_iXlinker.EtherCAT_Master_BKCUCX.TcTerminals210_EK1100_2.TcTerminals210_2BK1250.A_0006_KL_6211_ASI_Master_Parameter_Interface_and_16_Byte_31_ASI_Slaves_Power.Channel_1.ASI_In_Slave_23 <-> Channel 1/ASI In Slave 23
//     PlcTask Inputs/GVL_iXlinker.EtherCAT_Master_BKCUCX.TcTerminals210_EK1100_2.TcTerminals210_2BK1250.A_0006_KL_6211_ASI_Master_Parameter_Interface_and_16_Byte_31_ASI_Slaves_Power.Channel_1.ASI_In_Slave_24 <-> Channel 1/ASI In Slave 24
//     PlcTask Inputs/GVL_iXlinker.EtherCAT_Master_BKCUCX.TcTerminals210_EK1100_2.TcTerminals210_2BK1250.A_0006_KL_6211_ASI_Master_Parameter_Interface_and_16_Byte_31_ASI_Slaves_Power.Channel_1.ASI_In_Slave_25 <-> Channel 1/ASI In Slave 25
//     PlcTask Inputs/GVL_iXlinker.EtherCAT_Master_BKCUCX.TcTerminals210_EK1100_2.TcTerminals210_2BK1250.A_0006_KL_6211_ASI_Master_Parameter_Interface_and_16_Byte_31_ASI_Slaves_Power.Channel_1.ASI_In_Slave_26 <-> Channel 1/ASI In Slave 26
//     PlcTask Inputs/GVL_iXlinker.EtherCAT_Master_BKCUCX.TcTerminals210_EK1100_2.TcTerminals210_2BK1250.A_0006_KL_6211_ASI_Master_Parameter_Interface_and_16_Byte_31_ASI_Slaves_Power.Channel_1.ASI_In_Slave_27 <-> Channel 1/ASI In Slave 27
//     PlcTask Inputs/GVL_iXlinker.EtherCAT_Master_BKCUCX.TcTerminals210_EK1100_2.TcTerminals210_2BK1250.A_0006_KL_6211_ASI_Master_Parameter_Interface_and_16_Byte_31_ASI_Slaves_Power.Channel_1.ASI_In_Slave_28 <-> Channel 1/ASI In Slave 28
//     PlcTask Inputs/GVL_iXlinker.EtherCAT_Master_BKCUCX.TcTerminals210_EK1100_2.TcTerminals210_2BK1250.A_0006_KL_6211_ASI_Master_Parameter_Interface_and_16_Byte_31_ASI_Slaves_Power.Channel_1.ASI_In_Slave_29 <-> Channel 1/ASI In Slave 29
//     PlcTask Inputs/GVL_iXlinker.EtherCAT_Master_BKCUCX.TcTerminals210_EK1100_2.TcTerminals210_2BK1250.A_0006_KL_6211_ASI_Master_Parameter_Interface_and_16_Byte_31_ASI_Slaves_Power.Channel_1.ASI_In_Slave_30 <-> Channel 1/ASI In Slave 30
//     PlcTask Inputs/GVL_iXlinker.EtherCAT_Master_BKCUCX.TcTerminals210_EK1100_2.TcTerminals210_2BK1250.A_0006_KL_6211_ASI_Master_Parameter_Interface_and_16_Byte_31_ASI_Slaves_Power.Channel_1.ASI_In_Slave_31 <-> Channel 1/ASI In Slave 31
//     PlcTask Outputs/GVL_iXlinker.EtherCAT_Master_BKCUCX.TcTerminals210_EK1100_2.TcTerminals210_2BK1250.A_0006_KL_6211_ASI_Master_Parameter_Interface_and_16_Byte_31_ASI_Slaves_Power.Channel_1.Control <-> Channel 1/Control
//     PlcTask Outputs/GVL_iXlinker.EtherCAT_Master_BKCUCX.TcTerminals210_EK1100_2.TcTerminals210_2BK1250.A_0006_KL_6211_ASI_Master_Parameter_Interface_and_16_Byte_31_ASI_Slaves_Power.Channel_1.Parameter_Out <-> Channel 1/Parameter Out
//     PlcTask Outputs/GVL_iXlinker.EtherCAT_Master_BKCUCX.TcTerminals210_EK1100_2.TcTerminals210_2BK1250.A_0006_KL_6211_ASI_Master_Parameter_Interface_and_16_Byte_31_ASI_Slaves_Power.Channel_1.ASI_Out_Control <-> Channel 1/ASI Out Control
//     PlcTask Outputs/GVL_iXlinker.EtherCAT_Master_BKCUCX.TcTerminals210_EK1100_2.TcTerminals210_2BK1250.A_0006_KL_6211_ASI_Master_Parameter_Interface_and_16_Byte_31_ASI_Slaves_Power.Channel_1.ASI_Out_Slave_1 <-> Channel 1/ASI Out Slave 1
//     PlcTask Outputs/GVL_iXlinker.EtherCAT_Master_BKCUCX.TcTerminals210_EK1100_2.TcTerminals210_2BK1250.A_0006_KL_6211_ASI_Master_Parameter_Interface_and_16_Byte_31_ASI_Slaves_Power.Channel_1.ASI_Out_Slave_2 <-> Channel 1/ASI Out Slave 2
//     PlcTask Outputs/GVL_iXlinker.EtherCAT_Master_BKCUCX.TcTerminals210_EK1100_2.TcTerminals210_2BK1250.A_0006_KL_6211_ASI_Master_Parameter_Interface_and_16_Byte_31_ASI_Slaves_Power.Channel_1.ASI_Out_Slave_3 <-> Channel 1/ASI Out Slave 3
//     PlcTask Outputs/GVL_iXlinker.EtherCAT_Master_BKCUCX.TcTerminals210_EK1100_2.TcTerminals210_2BK1250.A_0006_KL_6211_ASI_Master_Parameter_Interface_and_16_Byte_31_ASI_Slaves_Power.Channel_1.ASI_Out_Slave_4 <-> Channel 1/ASI Out Slave 4
//     PlcTask Outputs/GVL_iXlinker.EtherCAT_Master_BKCUCX.TcTerminals210_EK1100_2.TcTerminals210_2BK1250.A_0006_KL_6211_ASI_Master_Parameter_Interface_and_16_Byte_31_ASI_Slaves_Power.Channel_1.ASI_Out_Slave_5 <-> Channel 1/ASI Out Slave 5
//     PlcTask Outputs/GVL_iXlinker.EtherCAT_Master_BKCUCX.TcTerminals210_EK1100_2.TcTerminals210_2BK1250.A_0006_KL_6211_ASI_Master_Parameter_Interface_and_16_Byte_31_ASI_Slaves_Power.Channel_1.ASI_Out_Slave_6 <-> Channel 1/ASI Out Slave 6
//     PlcTask Outputs/GVL_iXlinker.EtherCAT_Master_BKCUCX.TcTerminals210_EK1100_2.TcTerminals210_2BK1250.A_0006_KL_6211_ASI_Master_Parameter_Interface_and_16_Byte_31_ASI_Slaves_Power.Channel_1.ASI_Out_Slave_7 <-> Channel 1/ASI Out Slave 7
//     PlcTask Outputs/GVL_iXlinker.EtherCAT_Master_BKCUCX.TcTerminals210_EK1100_2.TcTerminals210_2BK1250.A_0006_KL_6211_ASI_Master_Parameter_Interface_and_16_Byte_31_ASI_Slaves_Power.Channel_1.ASI_Out_Slave_8 <-> Channel 1/ASI Out Slave 8
//     PlcTask Outputs/GVL_iXlinker.EtherCAT_Master_BKCUCX.TcTerminals210_EK1100_2.TcTerminals210_2BK1250.A_0006_KL_6211_ASI_Master_Parameter_Interface_and_16_Byte_31_ASI_Slaves_Power.Channel_1.ASI_Out_Slave_9 <-> Channel 1/ASI Out Slave 9
//     PlcTask Outputs/GVL_iXlinker.EtherCAT_Master_BKCUCX.TcTerminals210_EK1100_2.TcTerminals210_2BK1250.A_0006_KL_6211_ASI_Master_Parameter_Interface_and_16_Byte_31_ASI_Slaves_Power.Channel_1.ASI_Out_Slave_10 <-> Channel 1/ASI Out Slave 10
//     PlcTask Outputs/GVL_iXlinker.EtherCAT_Master_BKCUCX.TcTerminals210_EK1100_2.TcTerminals210_2BK1250.A_0006_KL_6211_ASI_Master_Parameter_Interface_and_16_Byte_31_ASI_Slaves_Power.Channel_1.ASI_Out_Slave_11 <-> Channel 1/ASI Out Slave 11
//     PlcTask Outputs/GVL_iXlinker.EtherCAT_Master_BKCUCX.TcTerminals210_EK1100_2.TcTerminals210_2BK1250.A_0006_KL_6211_ASI_Master_Parameter_Interface_and_16_Byte_31_ASI_Slaves_Power.Channel_1.ASI_Out_Slave_12 <-> Channel 1/ASI Out Slave 12
//     PlcTask Outputs/GVL_iXlinker.EtherCAT_Master_BKCUCX.TcTerminals210_EK1100_2.TcTerminals210_2BK1250.A_0006_KL_6211_ASI_Master_Parameter_Interface_and_16_Byte_31_ASI_Slaves_Power.Channel_1.ASI_Out_Slave_13 <-> Channel 1/ASI Out Slave 13
//     PlcTask Outputs/GVL_iXlinker.EtherCAT_Master_BKCUCX.TcTerminals210_EK1100_2.TcTerminals210_2BK1250.A_0006_KL_6211_ASI_Master_Parameter_Interface_and_16_Byte_31_ASI_Slaves_Power.Channel_1.ASI_Out_Slave_14 <-> Channel 1/ASI Out Slave 14
//     PlcTask Outputs/GVL_iXlinker.EtherCAT_Master_BKCUCX.TcTerminals210_EK1100_2.TcTerminals210_2BK1250.A_0006_KL_6211_ASI_Master_Parameter_Interface_and_16_Byte_31_ASI_Slaves_Power.Channel_1.ASI_Out_Slave_15 <-> Channel 1/ASI Out Slave 15
//     PlcTask Outputs/GVL_iXlinker.EtherCAT_Master_BKCUCX.TcTerminals210_EK1100_2.TcTerminals210_2BK1250.A_0006_KL_6211_ASI_Master_Parameter_Interface_and_16_Byte_31_ASI_Slaves_Power.Channel_1.ASI_Out_Slave_16 <-> Channel 1/ASI Out Slave 16
//     PlcTask Outputs/GVL_iXlinker.EtherCAT_Master_BKCUCX.TcTerminals210_EK1100_2.TcTerminals210_2BK1250.A_0006_KL_6211_ASI_Master_Parameter_Interface_and_16_Byte_31_ASI_Slaves_Power.Channel_1.ASI_Out_Slave_17 <-> Channel 1/ASI Out Slave 17
//     PlcTask Outputs/GVL_iXlinker.EtherCAT_Master_BKCUCX.TcTerminals210_EK1100_2.TcTerminals210_2BK1250.A_0006_KL_6211_ASI_Master_Parameter_Interface_and_16_Byte_31_ASI_Slaves_Power.Channel_1.ASI_Out_Slave_18 <-> Channel 1/ASI Out Slave 18
//     PlcTask Outputs/GVL_iXlinker.EtherCAT_Master_BKCUCX.TcTerminals210_EK1100_2.TcTerminals210_2BK1250.A_0006_KL_6211_ASI_Master_Parameter_Interface_and_16_Byte_31_ASI_Slaves_Power.Channel_1.ASI_Out_Slave_19 <-> Channel 1/ASI Out Slave 19
//     PlcTask Outputs/GVL_iXlinker.EtherCAT_Master_BKCUCX.TcTerminals210_EK1100_2.TcTerminals210_2BK1250.A_0006_KL_6211_ASI_Master_Parameter_Interface_and_16_Byte_31_ASI_Slaves_Power.Channel_1.ASI_Out_Slave_20 <-> Channel 1/ASI Out Slave 20
//     PlcTask Outputs/GVL_iXlinker.EtherCAT_Master_BKCUCX.TcTerminals210_EK1100_2.TcTerminals210_2BK1250.A_0006_KL_6211_ASI_Master_Parameter_Interface_and_16_Byte_31_ASI_Slaves_Power.Channel_1.ASI_Out_Slave_21 <-> Channel 1/ASI Out Slave 21
//     PlcTask Outputs/GVL_iXlinker.EtherCAT_Master_BKCUCX.TcTerminals210_EK1100_2.TcTerminals210_2BK1250.A_0006_KL_6211_ASI_Master_Parameter_Interface_and_16_Byte_31_ASI_Slaves_Power.Channel_1.ASI_Out_Slave_22 <-> Channel 1/ASI Out Slave 22
//     PlcTask Outputs/GVL_iXlinker.EtherCAT_Master_BKCUCX.TcTerminals210_EK1100_2.TcTerminals210_2BK1250.A_0006_KL_6211_ASI_Master_Parameter_Interface_and_16_Byte_31_ASI_Slaves_Power.Channel_1.ASI_Out_Slave_23 <-> Channel 1/ASI Out Slave 23
//     PlcTask Outputs/GVL_iXlinker.EtherCAT_Master_BKCUCX.TcTerminals210_EK1100_2.TcTerminals210_2BK1250.A_0006_KL_6211_ASI_Master_Parameter_Interface_and_16_Byte_31_ASI_Slaves_Power.Channel_1.ASI_Out_Slave_24 <-> Channel 1/ASI Out Slave 24
//     PlcTask Outputs/GVL_iXlinker.EtherCAT_Master_BKCUCX.TcTerminals210_EK1100_2.TcTerminals210_2BK1250.A_0006_KL_6211_ASI_Master_Parameter_Interface_and_16_Byte_31_ASI_Slaves_Power.Channel_1.ASI_Out_Slave_25 <-> Channel 1/ASI Out Slave 25
//     PlcTask Outputs/GVL_iXlinker.EtherCAT_Master_BKCUCX.TcTerminals210_EK1100_2.TcTerminals210_2BK1250.A_0006_KL_6211_ASI_Master_Parameter_Interface_and_16_Byte_31_ASI_Slaves_Power.Channel_1.ASI_Out_Slave_26 <-> Channel 1/ASI Out Slave 26
//     PlcTask Outputs/GVL_iXlinker.EtherCAT_Master_BKCUCX.TcTerminals210_EK1100_2.TcTerminals210_2BK1250.A_0006_KL_6211_ASI_Master_Parameter_Interface_and_16_Byte_31_ASI_Slaves_Power.Channel_1.ASI_Out_Slave_27 <-> Channel 1/ASI Out Slave 27
//     PlcTask Outputs/GVL_iXlinker.EtherCAT_Master_BKCUCX.TcTerminals210_EK1100_2.TcTerminals210_2BK1250.A_0006_KL_6211_ASI_Master_Parameter_Interface_and_16_Byte_31_ASI_Slaves_Power.Channel_1.ASI_Out_Slave_28 <-> Channel 1/ASI Out Slave 28
//     PlcTask Outputs/GVL_iXlinker.EtherCAT_Master_BKCUCX.TcTerminals210_EK1100_2.TcTerminals210_2BK1250.A_0006_KL_6211_ASI_Master_Parameter_Interface_and_16_Byte_31_ASI_Slaves_Power.Channel_1.ASI_Out_Slave_29 <-> Channel 1/ASI Out Slave 29
//     PlcTask Outputs/GVL_iXlinker.EtherCAT_Master_BKCUCX.TcTerminals210_EK1100_2.TcTerminals210_2BK1250.A_0006_KL_6211_ASI_Master_Parameter_Interface_and_16_Byte_31_ASI_Slaves_Power.Channel_1.ASI_Out_Slave_30 <-> Channel 1/ASI Out Slave 30
//     PlcTask Outputs/GVL_iXlinker.EtherCAT_Master_BKCUCX.TcTerminals210_EK1100_2.TcTerminals210_2BK1250.A_0006_KL_6211_ASI_Master_Parameter_Interface_and_16_Byte_31_ASI_Slaves_Power.Channel_1.ASI_Out_Slave_31 <-> Channel 1/ASI Out Slave 31
//   PLC/PLC Instance <-> EtherCAT Master BKCUCX/TcTerminals210_EK1100_2/TcTerminals210_2BK1250/A_0009(KL 6211 ASI-Master (Parameter Interface and 32 Byte (62 ASI-Slaves), Power))
//     PlcTask Inputs/GVL_iXlinker.EtherCAT_Master_BKCUCX.TcTerminals210_EK1100_2.TcTerminals210_2BK1250.A_0009_KL_6211_ASI_Master_Parameter_Interface_and_32_Byte_62_ASI_Slaves_Power.Channel_1.Status <-> Channel 1/Status
//     PlcTask Inputs/GVL_iXlinker.EtherCAT_Master_BKCUCX.TcTerminals210_EK1100_2.TcTerminals210_2BK1250.A_0009_KL_6211_ASI_Master_Parameter_Interface_and_32_Byte_62_ASI_Slaves_Power.Channel_1.Parameter_In <-> Channel 1/Parameter In
//     PlcTask Inputs/GVL_iXlinker.EtherCAT_Master_BKCUCX.TcTerminals210_EK1100_2.TcTerminals210_2BK1250.A_0009_KL_6211_ASI_Master_Parameter_Interface_and_32_Byte_62_ASI_Slaves_Power.Channel_1.ASI_In_Slave_1_Status <-> Channel 1/ASI In Slave 1 Status
//     PlcTask Inputs/GVL_iXlinker.EtherCAT_Master_BKCUCX.TcTerminals210_EK1100_2.TcTerminals210_2BK1250.A_0009_KL_6211_ASI_Master_Parameter_Interface_and_32_Byte_62_ASI_Slaves_Power.Channel_1.ASI_In_Slave_3_Slave_2 <-> Channel 1/ASI In Slave 3 Slave 2
//     PlcTask Inputs/GVL_iXlinker.EtherCAT_Master_BKCUCX.TcTerminals210_EK1100_2.TcTerminals210_2BK1250.A_0009_KL_6211_ASI_Master_Parameter_Interface_and_32_Byte_62_ASI_Slaves_Power.Channel_1.ASI_In_Slave_5_Slave_4 <-> Channel 1/ASI In Slave 5 Slave 4
//     PlcTask Inputs/GVL_iXlinker.EtherCAT_Master_BKCUCX.TcTerminals210_EK1100_2.TcTerminals210_2BK1250.A_0009_KL_6211_ASI_Master_Parameter_Interface_and_32_Byte_62_ASI_Slaves_Power.Channel_1.ASI_In_Slave_7_Slave_6 <-> Channel 1/ASI In Slave 7 Slave 6
//     PlcTask Inputs/GVL_iXlinker.EtherCAT_Master_BKCUCX.TcTerminals210_EK1100_2.TcTerminals210_2BK1250.A_0009_KL_6211_ASI_Master_Parameter_Interface_and_32_Byte_62_ASI_Slaves_Power.Channel_1.ASI_In_Slave_9_Slave_8 <-> Channel 1/ASI In Slave 9 Slave 8
//     PlcTask Inputs/GVL_iXlinker.EtherCAT_Master_BKCUCX.TcTerminals210_EK1100_2.TcTerminals210_2BK1250.A_0009_KL_6211_ASI_Master_Parameter_Interface_and_32_Byte_62_ASI_Slaves_Power.Channel_1.ASI_In_Slave_11_Slave_10 <-> Channel 1/ASI In Slave 11 Slave 10
//     PlcTask Inputs/GVL_iXlinker.EtherCAT_Master_BKCUCX.TcTerminals210_EK1100_2.TcTerminals210_2BK1250.A_0009_KL_6211_ASI_Master_Parameter_Interface_and_32_Byte_62_ASI_Slaves_Power.Channel_1.ASI_In_Slave_13_Slave_12 <-> Channel 1/ASI In Slave 13 Slave 12
//     PlcTask Inputs/GVL_iXlinker.EtherCAT_Master_BKCUCX.TcTerminals210_EK1100_2.TcTerminals210_2BK1250.A_0009_KL_6211_ASI_Master_Parameter_Interface_and_32_Byte_62_ASI_Slaves_Power.Channel_1.ASI_In_Slave_15_Slave_14 <-> Channel 1/ASI In Slave 15 Slave 14
//     PlcTask Inputs/GVL_iXlinker.EtherCAT_Master_BKCUCX.TcTerminals210_EK1100_2.TcTerminals210_2BK1250.A_0009_KL_6211_ASI_Master_Parameter_Interface_and_32_Byte_62_ASI_Slaves_Power.Channel_1.ASI_In_Slave_17_Slave_16 <-> Channel 1/ASI In Slave 17 Slave 16
//     PlcTask Inputs/GVL_iXlinker.EtherCAT_Master_BKCUCX.TcTerminals210_EK1100_2.TcTerminals210_2BK1250.A_0009_KL_6211_ASI_Master_Parameter_Interface_and_32_Byte_62_ASI_Slaves_Power.Channel_1.ASI_In_Slave_19_Slave_18 <-> Channel 1/ASI In Slave 19 Slave 18
//     PlcTask Inputs/GVL_iXlinker.EtherCAT_Master_BKCUCX.TcTerminals210_EK1100_2.TcTerminals210_2BK1250.A_0009_KL_6211_ASI_Master_Parameter_Interface_and_32_Byte_62_ASI_Slaves_Power.Channel_1.ASI_In_Slave_21_Slave_20 <-> Channel 1/ASI In Slave 21 Slave 20
//     PlcTask Inputs/GVL_iXlinker.EtherCAT_Master_BKCUCX.TcTerminals210_EK1100_2.TcTerminals210_2BK1250.A_0009_KL_6211_ASI_Master_Parameter_Interface_and_32_Byte_62_ASI_Slaves_Power.Channel_1.ASI_In_Slave_23_Slave_22 <-> Channel 1/ASI In Slave 23 Slave 22
//     PlcTask Inputs/GVL_iXlinker.EtherCAT_Master_BKCUCX.TcTerminals210_EK1100_2.TcTerminals210_2BK1250.A_0009_KL_6211_ASI_Master_Parameter_Interface_and_32_Byte_62_ASI_Slaves_Power.Channel_1.ASI_In_Slave_25_Slave_24 <-> Channel 1/ASI In Slave 25 Slave 24
//     PlcTask Inputs/GVL_iXlinker.EtherCAT_Master_BKCUCX.TcTerminals210_EK1100_2.TcTerminals210_2BK1250.A_0009_KL_6211_ASI_Master_Parameter_Interface_and_32_Byte_62_ASI_Slaves_Power.Channel_1.ASI_In_Slave_27_Slave_26 <-> Channel 1/ASI In Slave 27 Slave 26
//     PlcTask Inputs/GVL_iXlinker.EtherCAT_Master_BKCUCX.TcTerminals210_EK1100_2.TcTerminals210_2BK1250.A_0009_KL_6211_ASI_Master_Parameter_Interface_and_32_Byte_62_ASI_Slaves_Power.Channel_1.ASI_In_Slave_29_Slave_28 <-> Channel 1/ASI In Slave 29 Slave 28
//     PlcTask Inputs/GVL_iXlinker.EtherCAT_Master_BKCUCX.TcTerminals210_EK1100_2.TcTerminals210_2BK1250.A_0009_KL_6211_ASI_Master_Parameter_Interface_and_32_Byte_62_ASI_Slaves_Power.Channel_1.ASI_In_Slave_31_Slave_30 <-> Channel 1/ASI In Slave 31 Slave 30
//     PlcTask Inputs/GVL_iXlinker.EtherCAT_Master_BKCUCX.TcTerminals210_EK1100_2.TcTerminals210_2BK1250.A_0009_KL_6211_ASI_Master_Parameter_Interface_and_32_Byte_62_ASI_Slaves_Power.Channel_1.ASI_In_Slave_33_Slave_32 <-> Channel 1/ASI In Slave 33 Slave 32
//     PlcTask Inputs/GVL_iXlinker.EtherCAT_Master_BKCUCX.TcTerminals210_EK1100_2.TcTerminals210_2BK1250.A_0009_KL_6211_ASI_Master_Parameter_Interface_and_32_Byte_62_ASI_Slaves_Power.Channel_1.ASI_In_Slave_35_Slave_34 <-> Channel 1/ASI In Slave 35 Slave 34
//     PlcTask Inputs/GVL_iXlinker.EtherCAT_Master_BKCUCX.TcTerminals210_EK1100_2.TcTerminals210_2BK1250.A_0009_KL_6211_ASI_Master_Parameter_Interface_and_32_Byte_62_ASI_Slaves_Power.Channel_1.ASI_In_Slave_37_Slave_36 <-> Channel 1/ASI In Slave 37 Slave 36
//     PlcTask Inputs/GVL_iXlinker.EtherCAT_Master_BKCUCX.TcTerminals210_EK1100_2.TcTerminals210_2BK1250.A_0009_KL_6211_ASI_Master_Parameter_Interface_and_32_Byte_62_ASI_Slaves_Power.Channel_1.ASI_In_Slave_39_Slave_38 <-> Channel 1/ASI In Slave 39 Slave 38
//     PlcTask Inputs/GVL_iXlinker.EtherCAT_Master_BKCUCX.TcTerminals210_EK1100_2.TcTerminals210_2BK1250.A_0009_KL_6211_ASI_Master_Parameter_Interface_and_32_Byte_62_ASI_Slaves_Power.Channel_1.ASI_In_Slave_41_Slave_40 <-> Channel 1/ASI In Slave 41 Slave 40
//     PlcTask Inputs/GVL_iXlinker.EtherCAT_Master_BKCUCX.TcTerminals210_EK1100_2.TcTerminals210_2BK1250.A_0009_KL_6211_ASI_Master_Parameter_Interface_and_32_Byte_62_ASI_Slaves_Power.Channel_1.ASI_In_Slave_43_Slave_42 <-> Channel 1/ASI In Slave 43 Slave 42
//     PlcTask Inputs/GVL_iXlinker.EtherCAT_Master_BKCUCX.TcTerminals210_EK1100_2.TcTerminals210_2BK1250.A_0009_KL_6211_ASI_Master_Parameter_Interface_and_32_Byte_62_ASI_Slaves_Power.Channel_1.ASI_In_Slave_45_Slave_44 <-> Channel 1/ASI In Slave 45 Slave 44
//     PlcTask Inputs/GVL_iXlinker.EtherCAT_Master_BKCUCX.TcTerminals210_EK1100_2.TcTerminals210_2BK1250.A_0009_KL_6211_ASI_Master_Parameter_Interface_and_32_Byte_62_ASI_Slaves_Power.Channel_1.ASI_In_Slave_47_Slave_46 <-> Channel 1/ASI In Slave 47 Slave 46
//     PlcTask Inputs/GVL_iXlinker.EtherCAT_Master_BKCUCX.TcTerminals210_EK1100_2.TcTerminals210_2BK1250.A_0009_KL_6211_ASI_Master_Parameter_Interface_and_32_Byte_62_ASI_Slaves_Power.Channel_1.ASI_In_Slave_49_Slave_48 <-> Channel 1/ASI In Slave 49 Slave 48
//     PlcTask Inputs/GVL_iXlinker.EtherCAT_Master_BKCUCX.TcTerminals210_EK1100_2.TcTerminals210_2BK1250.A_0009_KL_6211_ASI_Master_Parameter_Interface_and_32_Byte_62_ASI_Slaves_Power.Channel_1.ASI_In_Slave_51_Slave_50 <-> Channel 1/ASI In Slave 51 Slave 50
//     PlcTask Inputs/GVL_iXlinker.EtherCAT_Master_BKCUCX.TcTerminals210_EK1100_2.TcTerminals210_2BK1250.A_0009_KL_6211_ASI_Master_Parameter_Interface_and_32_Byte_62_ASI_Slaves_Power.Channel_1.ASI_In_Slave_53_Slave_52 <-> Channel 1/ASI In Slave 53 Slave 52
//     PlcTask Inputs/GVL_iXlinker.EtherCAT_Master_BKCUCX.TcTerminals210_EK1100_2.TcTerminals210_2BK1250.A_0009_KL_6211_ASI_Master_Parameter_Interface_and_32_Byte_62_ASI_Slaves_Power.Channel_1.ASI_In_Slave_55_Slave_54 <-> Channel 1/ASI In Slave 55 Slave 54
//     PlcTask Inputs/GVL_iXlinker.EtherCAT_Master_BKCUCX.TcTerminals210_EK1100_2.TcTerminals210_2BK1250.A_0009_KL_6211_ASI_Master_Parameter_Interface_and_32_Byte_62_ASI_Slaves_Power.Channel_1.ASI_In_Slave_57_Slave_56 <-> Channel 1/ASI In Slave 57 Slave 56
//     PlcTask Inputs/GVL_iXlinker.EtherCAT_Master_BKCUCX.TcTerminals210_EK1100_2.TcTerminals210_2BK1250.A_0009_KL_6211_ASI_Master_Parameter_Interface_and_32_Byte_62_ASI_Slaves_Power.Channel_1.ASI_In_Slave_59_Slave_58 <-> Channel 1/ASI In Slave 59 Slave 58
//     PlcTask Inputs/GVL_iXlinker.EtherCAT_Master_BKCUCX.TcTerminals210_EK1100_2.TcTerminals210_2BK1250.A_0009_KL_6211_ASI_Master_Parameter_Interface_and_32_Byte_62_ASI_Slaves_Power.Channel_1.ASI_In_Slave_61_Slave_60 <-> Channel 1/ASI In Slave 61 Slave 60
//     PlcTask Inputs/GVL_iXlinker.EtherCAT_Master_BKCUCX.TcTerminals210_EK1100_2.TcTerminals210_2BK1250.A_0009_KL_6211_ASI_Master_Parameter_Interface_and_32_Byte_62_ASI_Slaves_Power.Channel_1.ASI_In_Slave_63_Slave_62 <-> Channel 1/ASI In Slave 63 Slave 62
//     PlcTask Outputs/GVL_iXlinker.EtherCAT_Master_BKCUCX.TcTerminals210_EK1100_2.TcTerminals210_2BK1250.A_0009_KL_6211_ASI_Master_Parameter_Interface_and_32_Byte_62_ASI_Slaves_Power.Channel_1.Control <-> Channel 1/Control
//     PlcTask Outputs/GVL_iXlinker.EtherCAT_Master_BKCUCX.TcTerminals210_EK1100_2.TcTerminals210_2BK1250.A_0009_KL_6211_ASI_Master_Parameter_Interface_and_32_Byte_62_ASI_Slaves_Power.Channel_1.Parameter_Out <-> Channel 1/Parameter Out
//     PlcTask Outputs/GVL_iXlinker.EtherCAT_Master_BKCUCX.TcTerminals210_EK1100_2.TcTerminals210_2BK1250.A_0009_KL_6211_ASI_Master_Parameter_Interface_and_32_Byte_62_ASI_Slaves_Power.Channel_1.ASI_Out_Slave_1_Control <-> Channel 1/ASI Out Slave 1 Control
//     PlcTask Outputs/GVL_iXlinker.EtherCAT_Master_BKCUCX.TcTerminals210_EK1100_2.TcTerminals210_2BK1250.A_0009_KL_6211_ASI_Master_Parameter_Interface_and_32_Byte_62_ASI_Slaves_Power.Channel_1.ASI_Out_Slave_3_Slave_2 <-> Channel 1/ASI Out Slave 3 Slave 2
//     PlcTask Outputs/GVL_iXlinker.EtherCAT_Master_BKCUCX.TcTerminals210_EK1100_2.TcTerminals210_2BK1250.A_0009_KL_6211_ASI_Master_Parameter_Interface_and_32_Byte_62_ASI_Slaves_Power.Channel_1.ASI_Out_Slave_5_Slave_4 <-> Channel 1/ASI Out Slave 5 Slave 4
//     PlcTask Outputs/GVL_iXlinker.EtherCAT_Master_BKCUCX.TcTerminals210_EK1100_2.TcTerminals210_2BK1250.A_0009_KL_6211_ASI_Master_Parameter_Interface_and_32_Byte_62_ASI_Slaves_Power.Channel_1.ASI_Out_Slave_7_Slave_6 <-> Channel 1/ASI Out Slave 7 Slave 6
//     PlcTask Outputs/GVL_iXlinker.EtherCAT_Master_BKCUCX.TcTerminals210_EK1100_2.TcTerminals210_2BK1250.A_0009_KL_6211_ASI_Master_Parameter_Interface_and_32_Byte_62_ASI_Slaves_Power.Channel_1.ASI_Out_Slave_9_Slave_8 <-> Channel 1/ASI Out Slave 9 Slave 8
//     PlcTask Outputs/GVL_iXlinker.EtherCAT_Master_BKCUCX.TcTerminals210_EK1100_2.TcTerminals210_2BK1250.A_0009_KL_6211_ASI_Master_Parameter_Interface_and_32_Byte_62_ASI_Slaves_Power.Channel_1.ASI_Out_Slave_11_Slave_10 <-> Channel 1/ASI Out Slave 11 Slave 10
//     PlcTask Outputs/GVL_iXlinker.EtherCAT_Master_BKCUCX.TcTerminals210_EK1100_2.TcTerminals210_2BK1250.A_0009_KL_6211_ASI_Master_Parameter_Interface_and_32_Byte_62_ASI_Slaves_Power.Channel_1.ASI_Out_Slave_13_Slave_12 <-> Channel 1/ASI Out Slave 13 Slave 12
//     PlcTask Outputs/GVL_iXlinker.EtherCAT_Master_BKCUCX.TcTerminals210_EK1100_2.TcTerminals210_2BK1250.A_0009_KL_6211_ASI_Master_Parameter_Interface_and_32_Byte_62_ASI_Slaves_Power.Channel_1.ASI_Out_Slave_15_Slave_14 <-> Channel 1/ASI Out Slave 15 Slave 14
//     PlcTask Outputs/GVL_iXlinker.EtherCAT_Master_BKCUCX.TcTerminals210_EK1100_2.TcTerminals210_2BK1250.A_0009_KL_6211_ASI_Master_Parameter_Interface_and_32_Byte_62_ASI_Slaves_Power.Channel_1.ASI_Out_Slave_17_Slave_16 <-> Channel 1/ASI Out Slave 17 Slave 16
//     PlcTask Outputs/GVL_iXlinker.EtherCAT_Master_BKCUCX.TcTerminals210_EK1100_2.TcTerminals210_2BK1250.A_0009_KL_6211_ASI_Master_Parameter_Interface_and_32_Byte_62_ASI_Slaves_Power.Channel_1.ASI_Out_Slave_19_Slave_18 <-> Channel 1/ASI Out Slave 19 Slave 18
//     PlcTask Outputs/GVL_iXlinker.EtherCAT_Master_BKCUCX.TcTerminals210_EK1100_2.TcTerminals210_2BK1250.A_0009_KL_6211_ASI_Master_Parameter_Interface_and_32_Byte_62_ASI_Slaves_Power.Channel_1.ASI_Out_Slave_21_Slave_20 <-> Channel 1/ASI Out Slave 21 Slave 20
//     PlcTask Outputs/GVL_iXlinker.EtherCAT_Master_BKCUCX.TcTerminals210_EK1100_2.TcTerminals210_2BK1250.A_0009_KL_6211_ASI_Master_Parameter_Interface_and_32_Byte_62_ASI_Slaves_Power.Channel_1.ASI_Out_Slave_23_Slave_22 <-> Channel 1/ASI Out Slave 23 Slave 22
//     PlcTask Outputs/GVL_iXlinker.EtherCAT_Master_BKCUCX.TcTerminals210_EK1100_2.TcTerminals210_2BK1250.A_0009_KL_6211_ASI_Master_Parameter_Interface_and_32_Byte_62_ASI_Slaves_Power.Channel_1.ASI_Out_Slave_25_Slave_24 <-> Channel 1/ASI Out Slave 25 Slave 24
//     PlcTask Outputs/GVL_iXlinker.EtherCAT_Master_BKCUCX.TcTerminals210_EK1100_2.TcTerminals210_2BK1250.A_0009_KL_6211_ASI_Master_Parameter_Interface_and_32_Byte_62_ASI_Slaves_Power.Channel_1.ASI_Out_Slave_27_Slave_26 <-> Channel 1/ASI Out Slave 27 Slave 26
//     PlcTask Outputs/GVL_iXlinker.EtherCAT_Master_BKCUCX.TcTerminals210_EK1100_2.TcTerminals210_2BK1250.A_0009_KL_6211_ASI_Master_Parameter_Interface_and_32_Byte_62_ASI_Slaves_Power.Channel_1.ASI_Out_Slave_29_Slave_28 <-> Channel 1/ASI Out Slave 29 Slave 28
//     PlcTask Outputs/GVL_iXlinker.EtherCAT_Master_BKCUCX.TcTerminals210_EK1100_2.TcTerminals210_2BK1250.A_0009_KL_6211_ASI_Master_Parameter_Interface_and_32_Byte_62_ASI_Slaves_Power.Channel_1.ASI_Out_Slave_31_Slave_30 <-> Channel 1/ASI Out Slave 31 Slave 30
//     PlcTask Outputs/GVL_iXlinker.EtherCAT_Master_BKCUCX.TcTerminals210_EK1100_2.TcTerminals210_2BK1250.A_0009_KL_6211_ASI_Master_Parameter_Interface_and_32_Byte_62_ASI_Slaves_Power.Channel_1.ASI_Out_Slave_33_Slave_32 <-> Channel 1/ASI Out Slave 33 Slave 32
//     PlcTask Outputs/GVL_iXlinker.EtherCAT_Master_BKCUCX.TcTerminals210_EK1100_2.TcTerminals210_2BK1250.A_0009_KL_6211_ASI_Master_Parameter_Interface_and_32_Byte_62_ASI_Slaves_Power.Channel_1.ASI_Out_Slave_35_Slave_34 <-> Channel 1/ASI Out Slave 35 Slave 34
//     PlcTask Outputs/GVL_iXlinker.EtherCAT_Master_BKCUCX.TcTerminals210_EK1100_2.TcTerminals210_2BK1250.A_0009_KL_6211_ASI_Master_Parameter_Interface_and_32_Byte_62_ASI_Slaves_Power.Channel_1.ASI_Out_Slave_37_Slave_36 <-> Channel 1/ASI Out Slave 37 Slave 36
//     PlcTask Outputs/GVL_iXlinker.EtherCAT_Master_BKCUCX.TcTerminals210_EK1100_2.TcTerminals210_2BK1250.A_0009_KL_6211_ASI_Master_Parameter_Interface_and_32_Byte_62_ASI_Slaves_Power.Channel_1.ASI_Out_Slave_39_Slave_38 <-> Channel 1/ASI Out Slave 39 Slave 38
//     PlcTask Outputs/GVL_iXlinker.EtherCAT_Master_BKCUCX.TcTerminals210_EK1100_2.TcTerminals210_2BK1250.A_0009_KL_6211_ASI_Master_Parameter_Interface_and_32_Byte_62_ASI_Slaves_Power.Channel_1.ASI_Out_Slave_41_Slave_40 <-> Channel 1/ASI Out Slave 41 Slave 40
//     PlcTask Outputs/GVL_iXlinker.EtherCAT_Master_BKCUCX.TcTerminals210_EK1100_2.TcTerminals210_2BK1250.A_0009_KL_6211_ASI_Master_Parameter_Interface_and_32_Byte_62_ASI_Slaves_Power.Channel_1.ASI_Out_Slave_43_Slave_42 <-> Channel 1/ASI Out Slave 43 Slave 42
//     PlcTask Outputs/GVL_iXlinker.EtherCAT_Master_BKCUCX.TcTerminals210_EK1100_2.TcTerminals210_2BK1250.A_0009_KL_6211_ASI_Master_Parameter_Interface_and_32_Byte_62_ASI_Slaves_Power.Channel_1.ASI_Out_Slave_45_Slave_44 <-> Channel 1/ASI Out Slave 45 Slave 44
//     PlcTask Outputs/GVL_iXlinker.EtherCAT_Master_BKCUCX.TcTerminals210_EK1100_2.TcTerminals210_2BK1250.A_0009_KL_6211_ASI_Master_Parameter_Interface_and_32_Byte_62_ASI_Slaves_Power.Channel_1.ASI_Out_Slave_47_Slave_46 <-> Channel 1/ASI Out Slave 47 Slave 46
//     PlcTask Outputs/GVL_iXlinker.EtherCAT_Master_BKCUCX.TcTerminals210_EK1100_2.TcTerminals210_2BK1250.A_0009_KL_6211_ASI_Master_Parameter_Interface_and_32_Byte_62_ASI_Slaves_Power.Channel_1.ASI_Out_Slave_49_Slave_48 <-> Channel 1/ASI Out Slave 49 Slave 48
//     PlcTask Outputs/GVL_iXlinker.EtherCAT_Master_BKCUCX.TcTerminals210_EK1100_2.TcTerminals210_2BK1250.A_0009_KL_6211_ASI_Master_Parameter_Interface_and_32_Byte_62_ASI_Slaves_Power.Channel_1.ASI_Out_Slave_51_Slave_50 <-> Channel 1/ASI Out Slave 51 Slave 50
//     PlcTask Outputs/GVL_iXlinker.EtherCAT_Master_BKCUCX.TcTerminals210_EK1100_2.TcTerminals210_2BK1250.A_0009_KL_6211_ASI_Master_Parameter_Interface_and_32_Byte_62_ASI_Slaves_Power.Channel_1.ASI_Out_Slave_53_Slave_52 <-> Channel 1/ASI Out Slave 53 Slave 52
//     PlcTask Outputs/GVL_iXlinker.EtherCAT_Master_BKCUCX.TcTerminals210_EK1100_2.TcTerminals210_2BK1250.A_0009_KL_6211_ASI_Master_Parameter_Interface_and_32_Byte_62_ASI_Slaves_Power.Channel_1.ASI_Out_Slave_55_Slave_54 <-> Channel 1/ASI Out Slave 55 Slave 54
//     PlcTask Outputs/GVL_iXlinker.EtherCAT_Master_BKCUCX.TcTerminals210_EK1100_2.TcTerminals210_2BK1250.A_0009_KL_6211_ASI_Master_Parameter_Interface_and_32_Byte_62_ASI_Slaves_Power.Channel_1.ASI_Out_Slave_57_Slave_56 <-> Channel 1/ASI Out Slave 57 Slave 56
//     PlcTask Outputs/GVL_iXlinker.EtherCAT_Master_BKCUCX.TcTerminals210_EK1100_2.TcTerminals210_2BK1250.A_0009_KL_6211_ASI_Master_Parameter_Interface_and_32_Byte_62_ASI_Slaves_Power.Channel_1.ASI_Out_Slave_59_Slave_58 <-> Channel 1/ASI Out Slave 59 Slave 58
//     PlcTask Outputs/GVL_iXlinker.EtherCAT_Master_BKCUCX.TcTerminals210_EK1100_2.TcTerminals210_2BK1250.A_0009_KL_6211_ASI_Master_Parameter_Interface_and_32_Byte_62_ASI_Slaves_Power.Channel_1.ASI_Out_Slave_61_Slave_60 <-> Channel 1/ASI Out Slave 61 Slave 60
//     PlcTask Outputs/GVL_iXlinker.EtherCAT_Master_BKCUCX.TcTerminals210_EK1100_2.TcTerminals210_2BK1250.A_0009_KL_6211_ASI_Master_Parameter_Interface_and_32_Byte_62_ASI_Slaves_Power.Channel_1.ASI_Out_Slave_63_Slave_62 <-> Channel 1/ASI Out Slave 63 Slave 62
//   PLC/PLC Instance <-> EtherCAT Master BKCUCX/TcTerminals210_EK1100_2/TcTerminals210_2BK1250/A_0010(KL 6211 ASI-Master (Parameter Interface and 32 Byte (62 ASI-Slaves), Power))
//     PlcTask Inputs/GVL_iXlinker.EtherCAT_Master_BKCUCX.TcTerminals210_EK1100_2.TcTerminals210_2BK1250.A_0010_KL_6211_ASI_Master_Parameter_Interface_and_32_Byte_62_ASI_Slaves_Power.Channel_1.Status <-> Channel 1/Status
//     PlcTask Inputs/GVL_iXlinker.EtherCAT_Master_BKCUCX.TcTerminals210_EK1100_2.TcTerminals210_2BK1250.A_0010_KL_6211_ASI_Master_Parameter_Interface_and_32_Byte_62_ASI_Slaves_Power.Channel_1.Parameter_In <-> Channel 1/Parameter In
//     PlcTask Inputs/GVL_iXlinker.EtherCAT_Master_BKCUCX.TcTerminals210_EK1100_2.TcTerminals210_2BK1250.A_0010_KL_6211_ASI_Master_Parameter_Interface_and_32_Byte_62_ASI_Slaves_Power.Channel_1.ASI_In_Status <-> Channel 1/ASI In Status
//     PlcTask Inputs/GVL_iXlinker.EtherCAT_Master_BKCUCX.TcTerminals210_EK1100_2.TcTerminals210_2BK1250.A_0010_KL_6211_ASI_Master_Parameter_Interface_and_32_Byte_62_ASI_Slaves_Power.Channel_1.ASI_In_Slave_1 <-> Channel 1/ASI In Slave 1
//     PlcTask Inputs/GVL_iXlinker.EtherCAT_Master_BKCUCX.TcTerminals210_EK1100_2.TcTerminals210_2BK1250.A_0010_KL_6211_ASI_Master_Parameter_Interface_and_32_Byte_62_ASI_Slaves_Power.Channel_1.ASI_In_Slave_2 <-> Channel 1/ASI In Slave 2
//     PlcTask Inputs/GVL_iXlinker.EtherCAT_Master_BKCUCX.TcTerminals210_EK1100_2.TcTerminals210_2BK1250.A_0010_KL_6211_ASI_Master_Parameter_Interface_and_32_Byte_62_ASI_Slaves_Power.Channel_1.ASI_In_Slave_3 <-> Channel 1/ASI In Slave 3
//     PlcTask Inputs/GVL_iXlinker.EtherCAT_Master_BKCUCX.TcTerminals210_EK1100_2.TcTerminals210_2BK1250.A_0010_KL_6211_ASI_Master_Parameter_Interface_and_32_Byte_62_ASI_Slaves_Power.Channel_1.ASI_In_Slave_4 <-> Channel 1/ASI In Slave 4
//     PlcTask Inputs/GVL_iXlinker.EtherCAT_Master_BKCUCX.TcTerminals210_EK1100_2.TcTerminals210_2BK1250.A_0010_KL_6211_ASI_Master_Parameter_Interface_and_32_Byte_62_ASI_Slaves_Power.Channel_1.ASI_In_Slave_5 <-> Channel 1/ASI In Slave 5
//     PlcTask Inputs/GVL_iXlinker.EtherCAT_Master_BKCUCX.TcTerminals210_EK1100_2.TcTerminals210_2BK1250.A_0010_KL_6211_ASI_Master_Parameter_Interface_and_32_Byte_62_ASI_Slaves_Power.Channel_1.ASI_In_Slave_6 <-> Channel 1/ASI In Slave 6
//     PlcTask Inputs/GVL_iXlinker.EtherCAT_Master_BKCUCX.TcTerminals210_EK1100_2.TcTerminals210_2BK1250.A_0010_KL_6211_ASI_Master_Parameter_Interface_and_32_Byte_62_ASI_Slaves_Power.Channel_1.ASI_In_Slave_7 <-> Channel 1/ASI In Slave 7
//     PlcTask Inputs/GVL_iXlinker.EtherCAT_Master_BKCUCX.TcTerminals210_EK1100_2.TcTerminals210_2BK1250.A_0010_KL_6211_ASI_Master_Parameter_Interface_and_32_Byte_62_ASI_Slaves_Power.Channel_1.ASI_In_Slave_8 <-> Channel 1/ASI In Slave 8
//     PlcTask Inputs/GVL_iXlinker.EtherCAT_Master_BKCUCX.TcTerminals210_EK1100_2.TcTerminals210_2BK1250.A_0010_KL_6211_ASI_Master_Parameter_Interface_and_32_Byte_62_ASI_Slaves_Power.Channel_1.ASI_In_Slave_9 <-> Channel 1/ASI In Slave 9
//     PlcTask Inputs/GVL_iXlinker.EtherCAT_Master_BKCUCX.TcTerminals210_EK1100_2.TcTerminals210_2BK1250.A_0010_KL_6211_ASI_Master_Parameter_Interface_and_32_Byte_62_ASI_Slaves_Power.Channel_1.ASI_In_Slave_10 <-> Channel 1/ASI In Slave 10
//     PlcTask Inputs/GVL_iXlinker.EtherCAT_Master_BKCUCX.TcTerminals210_EK1100_2.TcTerminals210_2BK1250.A_0010_KL_6211_ASI_Master_Parameter_Interface_and_32_Byte_62_ASI_Slaves_Power.Channel_1.ASI_In_Slave_11 <-> Channel 1/ASI In Slave 11
//     PlcTask Inputs/GVL_iXlinker.EtherCAT_Master_BKCUCX.TcTerminals210_EK1100_2.TcTerminals210_2BK1250.A_0010_KL_6211_ASI_Master_Parameter_Interface_and_32_Byte_62_ASI_Slaves_Power.Channel_1.ASI_In_Slave_12 <-> Channel 1/ASI In Slave 12
//     PlcTask Inputs/GVL_iXlinker.EtherCAT_Master_BKCUCX.TcTerminals210_EK1100_2.TcTerminals210_2BK1250.A_0010_KL_6211_ASI_Master_Parameter_Interface_and_32_Byte_62_ASI_Slaves_Power.Channel_1.ASI_In_Slave_13 <-> Channel 1/ASI In Slave 13
//     PlcTask Inputs/GVL_iXlinker.EtherCAT_Master_BKCUCX.TcTerminals210_EK1100_2.TcTerminals210_2BK1250.A_0010_KL_6211_ASI_Master_Parameter_Interface_and_32_Byte_62_ASI_Slaves_Power.Channel_1.ASI_In_Slave_14 <-> Channel 1/ASI In Slave 14
//     PlcTask Inputs/GVL_iXlinker.EtherCAT_Master_BKCUCX.TcTerminals210_EK1100_2.TcTerminals210_2BK1250.A_0010_KL_6211_ASI_Master_Parameter_Interface_and_32_Byte_62_ASI_Slaves_Power.Channel_1.ASI_In_Slave_15 <-> Channel 1/ASI In Slave 15
//     PlcTask Inputs/GVL_iXlinker.EtherCAT_Master_BKCUCX.TcTerminals210_EK1100_2.TcTerminals210_2BK1250.A_0010_KL_6211_ASI_Master_Parameter_Interface_and_32_Byte_62_ASI_Slaves_Power.Channel_1.ASI_In_Slave_16 <-> Channel 1/ASI In Slave 16
//     PlcTask Inputs/GVL_iXlinker.EtherCAT_Master_BKCUCX.TcTerminals210_EK1100_2.TcTerminals210_2BK1250.A_0010_KL_6211_ASI_Master_Parameter_Interface_and_32_Byte_62_ASI_Slaves_Power.Channel_1.ASI_In_Slave_17 <-> Channel 1/ASI In Slave 17
//     PlcTask Inputs/GVL_iXlinker.EtherCAT_Master_BKCUCX.TcTerminals210_EK1100_2.TcTerminals210_2BK1250.A_0010_KL_6211_ASI_Master_Parameter_Interface_and_32_Byte_62_ASI_Slaves_Power.Channel_1.ASI_In_Slave_18 <-> Channel 1/ASI In Slave 18
//     PlcTask Inputs/GVL_iXlinker.EtherCAT_Master_BKCUCX.TcTerminals210_EK1100_2.TcTerminals210_2BK1250.A_0010_KL_6211_ASI_Master_Parameter_Interface_and_32_Byte_62_ASI_Slaves_Power.Channel_1.ASI_In_Slave_19 <-> Channel 1/ASI In Slave 19
//     PlcTask Inputs/GVL_iXlinker.EtherCAT_Master_BKCUCX.TcTerminals210_EK1100_2.TcTerminals210_2BK1250.A_0010_KL_6211_ASI_Master_Parameter_Interface_and_32_Byte_62_ASI_Slaves_Power.Channel_1.ASI_In_Slave_20 <-> Channel 1/ASI In Slave 20
//     PlcTask Inputs/GVL_iXlinker.EtherCAT_Master_BKCUCX.TcTerminals210_EK1100_2.TcTerminals210_2BK1250.A_0010_KL_6211_ASI_Master_Parameter_Interface_and_32_Byte_62_ASI_Slaves_Power.Channel_1.ASI_In_Slave_21 <-> Channel 1/ASI In Slave 21
//     PlcTask Inputs/GVL_iXlinker.EtherCAT_Master_BKCUCX.TcTerminals210_EK1100_2.TcTerminals210_2BK1250.A_0010_KL_6211_ASI_Master_Parameter_Interface_and_32_Byte_62_ASI_Slaves_Power.Channel_1.ASI_In_Slave_22 <-> Channel 1/ASI In Slave 22
//     PlcTask Inputs/GVL_iXlinker.EtherCAT_Master_BKCUCX.TcTerminals210_EK1100_2.TcTerminals210_2BK1250.A_0010_KL_6211_ASI_Master_Parameter_Interface_and_32_Byte_62_ASI_Slaves_Power.Channel_1.ASI_In_Slave_23 <-> Channel 1/ASI In Slave 23
//     PlcTask Inputs/GVL_iXlinker.EtherCAT_Master_BKCUCX.TcTerminals210_EK1100_2.TcTerminals210_2BK1250.A_0010_KL_6211_ASI_Master_Parameter_Interface_and_32_Byte_62_ASI_Slaves_Power.Channel_1.ASI_In_Slave_24 <-> Channel 1/ASI In Slave 24
//     PlcTask Inputs/GVL_iXlinker.EtherCAT_Master_BKCUCX.TcTerminals210_EK1100_2.TcTerminals210_2BK1250.A_0010_KL_6211_ASI_Master_Parameter_Interface_and_32_Byte_62_ASI_Slaves_Power.Channel_1.ASI_In_Slave_25 <-> Channel 1/ASI In Slave 25
//     PlcTask Inputs/GVL_iXlinker.EtherCAT_Master_BKCUCX.TcTerminals210_EK1100_2.TcTerminals210_2BK1250.A_0010_KL_6211_ASI_Master_Parameter_Interface_and_32_Byte_62_ASI_Slaves_Power.Channel_1.ASI_In_Slave_26 <-> Channel 1/ASI In Slave 26
//     PlcTask Inputs/GVL_iXlinker.EtherCAT_Master_BKCUCX.TcTerminals210_EK1100_2.TcTerminals210_2BK1250.A_0010_KL_6211_ASI_Master_Parameter_Interface_and_32_Byte_62_ASI_Slaves_Power.Channel_1.ASI_In_Slave_27 <-> Channel 1/ASI In Slave 27
//     PlcTask Inputs/GVL_iXlinker.EtherCAT_Master_BKCUCX.TcTerminals210_EK1100_2.TcTerminals210_2BK1250.A_0010_KL_6211_ASI_Master_Parameter_Interface_and_32_Byte_62_ASI_Slaves_Power.Channel_1.ASI_In_Slave_28 <-> Channel 1/ASI In Slave 28
//     PlcTask Inputs/GVL_iXlinker.EtherCAT_Master_BKCUCX.TcTerminals210_EK1100_2.TcTerminals210_2BK1250.A_0010_KL_6211_ASI_Master_Parameter_Interface_and_32_Byte_62_ASI_Slaves_Power.Channel_1.ASI_In_Slave_29 <-> Channel 1/ASI In Slave 29
//     PlcTask Inputs/GVL_iXlinker.EtherCAT_Master_BKCUCX.TcTerminals210_EK1100_2.TcTerminals210_2BK1250.A_0010_KL_6211_ASI_Master_Parameter_Interface_and_32_Byte_62_ASI_Slaves_Power.Channel_1.ASI_In_Slave_30 <-> Channel 1/ASI In Slave 30
//     PlcTask Inputs/GVL_iXlinker.EtherCAT_Master_BKCUCX.TcTerminals210_EK1100_2.TcTerminals210_2BK1250.A_0010_KL_6211_ASI_Master_Parameter_Interface_and_32_Byte_62_ASI_Slaves_Power.Channel_1.ASI_In_Slave_31 <-> Channel 1/ASI In Slave 31
//     PlcTask Inputs/GVL_iXlinker.EtherCAT_Master_BKCUCX.TcTerminals210_EK1100_2.TcTerminals210_2BK1250.A_0010_KL_6211_ASI_Master_Parameter_Interface_and_32_Byte_62_ASI_Slaves_Power.Channel_1.ASI_In_Slave_32 <-> Channel 1/ASI In Slave 32
//     PlcTask Inputs/GVL_iXlinker.EtherCAT_Master_BKCUCX.TcTerminals210_EK1100_2.TcTerminals210_2BK1250.A_0010_KL_6211_ASI_Master_Parameter_Interface_and_32_Byte_62_ASI_Slaves_Power.Channel_1.ASI_In_Slave_33 <-> Channel 1/ASI In Slave 33
//     PlcTask Inputs/GVL_iXlinker.EtherCAT_Master_BKCUCX.TcTerminals210_EK1100_2.TcTerminals210_2BK1250.A_0010_KL_6211_ASI_Master_Parameter_Interface_and_32_Byte_62_ASI_Slaves_Power.Channel_1.ASI_In_Slave_34 <-> Channel 1/ASI In Slave 34
//     PlcTask Inputs/GVL_iXlinker.EtherCAT_Master_BKCUCX.TcTerminals210_EK1100_2.TcTerminals210_2BK1250.A_0010_KL_6211_ASI_Master_Parameter_Interface_and_32_Byte_62_ASI_Slaves_Power.Channel_1.ASI_In_Slave_35 <-> Channel 1/ASI In Slave 35
//     PlcTask Inputs/GVL_iXlinker.EtherCAT_Master_BKCUCX.TcTerminals210_EK1100_2.TcTerminals210_2BK1250.A_0010_KL_6211_ASI_Master_Parameter_Interface_and_32_Byte_62_ASI_Slaves_Power.Channel_1.ASI_In_Slave_36 <-> Channel 1/ASI In Slave 36
//     PlcTask Inputs/GVL_iXlinker.EtherCAT_Master_BKCUCX.TcTerminals210_EK1100_2.TcTerminals210_2BK1250.A_0010_KL_6211_ASI_Master_Parameter_Interface_and_32_Byte_62_ASI_Slaves_Power.Channel_1.ASI_In_Slave_37 <-> Channel 1/ASI In Slave 37
//     PlcTask Inputs/GVL_iXlinker.EtherCAT_Master_BKCUCX.TcTerminals210_EK1100_2.TcTerminals210_2BK1250.A_0010_KL_6211_ASI_Master_Parameter_Interface_and_32_Byte_62_ASI_Slaves_Power.Channel_1.ASI_In_Slave_38 <-> Channel 1/ASI In Slave 38
//     PlcTask Inputs/GVL_iXlinker.EtherCAT_Master_BKCUCX.TcTerminals210_EK1100_2.TcTerminals210_2BK1250.A_0010_KL_6211_ASI_Master_Parameter_Interface_and_32_Byte_62_ASI_Slaves_Power.Channel_1.ASI_In_Slave_39 <-> Channel 1/ASI In Slave 39
//     PlcTask Inputs/GVL_iXlinker.EtherCAT_Master_BKCUCX.TcTerminals210_EK1100_2.TcTerminals210_2BK1250.A_0010_KL_6211_ASI_Master_Parameter_Interface_and_32_Byte_62_ASI_Slaves_Power.Channel_1.ASI_In_Slave_40 <-> Channel 1/ASI In Slave 40
//     PlcTask Inputs/GVL_iXlinker.EtherCAT_Master_BKCUCX.TcTerminals210_EK1100_2.TcTerminals210_2BK1250.A_0010_KL_6211_ASI_Master_Parameter_Interface_and_32_Byte_62_ASI_Slaves_Power.Channel_1.ASI_In_Slave_41 <-> Channel 1/ASI In Slave 41
//     PlcTask Inputs/GVL_iXlinker.EtherCAT_Master_BKCUCX.TcTerminals210_EK1100_2.TcTerminals210_2BK1250.A_0010_KL_6211_ASI_Master_Parameter_Interface_and_32_Byte_62_ASI_Slaves_Power.Channel_1.ASI_In_Slave_42 <-> Channel 1/ASI In Slave 42
//     PlcTask Inputs/GVL_iXlinker.EtherCAT_Master_BKCUCX.TcTerminals210_EK1100_2.TcTerminals210_2BK1250.A_0010_KL_6211_ASI_Master_Parameter_Interface_and_32_Byte_62_ASI_Slaves_Power.Channel_1.ASI_In_Slave_43 <-> Channel 1/ASI In Slave 43
//     PlcTask Inputs/GVL_iXlinker.EtherCAT_Master_BKCUCX.TcTerminals210_EK1100_2.TcTerminals210_2BK1250.A_0010_KL_6211_ASI_Master_Parameter_Interface_and_32_Byte_62_ASI_Slaves_Power.Channel_1.ASI_In_Slave_44 <-> Channel 1/ASI In Slave 44
//     PlcTask Inputs/GVL_iXlinker.EtherCAT_Master_BKCUCX.TcTerminals210_EK1100_2.TcTerminals210_2BK1250.A_0010_KL_6211_ASI_Master_Parameter_Interface_and_32_Byte_62_ASI_Slaves_Power.Channel_1.ASI_In_Slave_45 <-> Channel 1/ASI In Slave 45
//     PlcTask Inputs/GVL_iXlinker.EtherCAT_Master_BKCUCX.TcTerminals210_EK1100_2.TcTerminals210_2BK1250.A_0010_KL_6211_ASI_Master_Parameter_Interface_and_32_Byte_62_ASI_Slaves_Power.Channel_1.ASI_In_Slave_46 <-> Channel 1/ASI In Slave 46
//     PlcTask Inputs/GVL_iXlinker.EtherCAT_Master_BKCUCX.TcTerminals210_EK1100_2.TcTerminals210_2BK1250.A_0010_KL_6211_ASI_Master_Parameter_Interface_and_32_Byte_62_ASI_Slaves_Power.Channel_1.ASI_In_Slave_47 <-> Channel 1/ASI In Slave 47
//     PlcTask Inputs/GVL_iXlinker.EtherCAT_Master_BKCUCX.TcTerminals210_EK1100_2.TcTerminals210_2BK1250.A_0010_KL_6211_ASI_Master_Parameter_Interface_and_32_Byte_62_ASI_Slaves_Power.Channel_1.ASI_In_Slave_48 <-> Channel 1/ASI In Slave 48
//     PlcTask Inputs/GVL_iXlinker.EtherCAT_Master_BKCUCX.TcTerminals210_EK1100_2.TcTerminals210_2BK1250.A_0010_KL_6211_ASI_Master_Parameter_Interface_and_32_Byte_62_ASI_Slaves_Power.Channel_1.ASI_In_Slave_49 <-> Channel 1/ASI In Slave 49
//     PlcTask Inputs/GVL_iXlinker.EtherCAT_Master_BKCUCX.TcTerminals210_EK1100_2.TcTerminals210_2BK1250.A_0010_KL_6211_ASI_Master_Parameter_Interface_and_32_Byte_62_ASI_Slaves_Power.Channel_1.ASI_In_Slave_50 <-> Channel 1/ASI In Slave 50
//     PlcTask Inputs/GVL_iXlinker.EtherCAT_Master_BKCUCX.TcTerminals210_EK1100_2.TcTerminals210_2BK1250.A_0010_KL_6211_ASI_Master_Parameter_Interface_and_32_Byte_62_ASI_Slaves_Power.Channel_1.ASI_In_Slave_51 <-> Channel 1/ASI In Slave 51
//     PlcTask Inputs/GVL_iXlinker.EtherCAT_Master_BKCUCX.TcTerminals210_EK1100_2.TcTerminals210_2BK1250.A_0010_KL_6211_ASI_Master_Parameter_Interface_and_32_Byte_62_ASI_Slaves_Power.Channel_1.ASI_In_Slave_52 <-> Channel 1/ASI In Slave 52
//     PlcTask Inputs/GVL_iXlinker.EtherCAT_Master_BKCUCX.TcTerminals210_EK1100_2.TcTerminals210_2BK1250.A_0010_KL_6211_ASI_Master_Parameter_Interface_and_32_Byte_62_ASI_Slaves_Power.Channel_1.ASI_In_Slave_53 <-> Channel 1/ASI In Slave 53
//     PlcTask Inputs/GVL_iXlinker.EtherCAT_Master_BKCUCX.TcTerminals210_EK1100_2.TcTerminals210_2BK1250.A_0010_KL_6211_ASI_Master_Parameter_Interface_and_32_Byte_62_ASI_Slaves_Power.Channel_1.ASI_In_Slave_54 <-> Channel 1/ASI In Slave 54
//     PlcTask Inputs/GVL_iXlinker.EtherCAT_Master_BKCUCX.TcTerminals210_EK1100_2.TcTerminals210_2BK1250.A_0010_KL_6211_ASI_Master_Parameter_Interface_and_32_Byte_62_ASI_Slaves_Power.Channel_1.ASI_In_Slave_55 <-> Channel 1/ASI In Slave 55
//     PlcTask Inputs/GVL_iXlinker.EtherCAT_Master_BKCUCX.TcTerminals210_EK1100_2.TcTerminals210_2BK1250.A_0010_KL_6211_ASI_Master_Parameter_Interface_and_32_Byte_62_ASI_Slaves_Power.Channel_1.ASI_In_Slave_56 <-> Channel 1/ASI In Slave 56
//     PlcTask Inputs/GVL_iXlinker.EtherCAT_Master_BKCUCX.TcTerminals210_EK1100_2.TcTerminals210_2BK1250.A_0010_KL_6211_ASI_Master_Parameter_Interface_and_32_Byte_62_ASI_Slaves_Power.Channel_1.ASI_In_Slave_57 <-> Channel 1/ASI In Slave 57
//     PlcTask Inputs/GVL_iXlinker.EtherCAT_Master_BKCUCX.TcTerminals210_EK1100_2.TcTerminals210_2BK1250.A_0010_KL_6211_ASI_Master_Parameter_Interface_and_32_Byte_62_ASI_Slaves_Power.Channel_1.ASI_In_Slave_58 <-> Channel 1/ASI In Slave 58
//     PlcTask Inputs/GVL_iXlinker.EtherCAT_Master_BKCUCX.TcTerminals210_EK1100_2.TcTerminals210_2BK1250.A_0010_KL_6211_ASI_Master_Parameter_Interface_and_32_Byte_62_ASI_Slaves_Power.Channel_1.ASI_In_Slave_59 <-> Channel 1/ASI In Slave 59
//     PlcTask Inputs/GVL_iXlinker.EtherCAT_Master_BKCUCX.TcTerminals210_EK1100_2.TcTerminals210_2BK1250.A_0010_KL_6211_ASI_Master_Parameter_Interface_and_32_Byte_62_ASI_Slaves_Power.Channel_1.ASI_In_Slave_60 <-> Channel 1/ASI In Slave 60
//     PlcTask Inputs/GVL_iXlinker.EtherCAT_Master_BKCUCX.TcTerminals210_EK1100_2.TcTerminals210_2BK1250.A_0010_KL_6211_ASI_Master_Parameter_Interface_and_32_Byte_62_ASI_Slaves_Power.Channel_1.ASI_In_Slave_61 <-> Channel 1/ASI In Slave 61
//     PlcTask Inputs/GVL_iXlinker.EtherCAT_Master_BKCUCX.TcTerminals210_EK1100_2.TcTerminals210_2BK1250.A_0010_KL_6211_ASI_Master_Parameter_Interface_and_32_Byte_62_ASI_Slaves_Power.Channel_1.ASI_In_Slave_62 <-> Channel 1/ASI In Slave 62
//     PlcTask Inputs/GVL_iXlinker.EtherCAT_Master_BKCUCX.TcTerminals210_EK1100_2.TcTerminals210_2BK1250.A_0010_KL_6211_ASI_Master_Parameter_Interface_and_32_Byte_62_ASI_Slaves_Power.Channel_1.ASI_In_Slave_63 <-> Channel 1/ASI In Slave 63
//     PlcTask Outputs/GVL_iXlinker.EtherCAT_Master_BKCUCX.TcTerminals210_EK1100_2.TcTerminals210_2BK1250.A_0010_KL_6211_ASI_Master_Parameter_Interface_and_32_Byte_62_ASI_Slaves_Power.Channel_1.Control <-> Channel 1/Control
//     PlcTask Outputs/GVL_iXlinker.EtherCAT_Master_BKCUCX.TcTerminals210_EK1100_2.TcTerminals210_2BK1250.A_0010_KL_6211_ASI_Master_Parameter_Interface_and_32_Byte_62_ASI_Slaves_Power.Channel_1.Parameter_Out <-> Channel 1/Parameter Out
//     PlcTask Outputs/GVL_iXlinker.EtherCAT_Master_BKCUCX.TcTerminals210_EK1100_2.TcTerminals210_2BK1250.A_0010_KL_6211_ASI_Master_Parameter_Interface_and_32_Byte_62_ASI_Slaves_Power.Channel_1.ASI_Out_Control <-> Channel 1/ASI Out Control
//     PlcTask Outputs/GVL_iXlinker.EtherCAT_Master_BKCUCX.TcTerminals210_EK1100_2.TcTerminals210_2BK1250.A_0010_KL_6211_ASI_Master_Parameter_Interface_and_32_Byte_62_ASI_Slaves_Power.Channel_1.ASI_Out_Slave_1 <-> Channel 1/ASI Out Slave 1
//     PlcTask Outputs/GVL_iXlinker.EtherCAT_Master_BKCUCX.TcTerminals210_EK1100_2.TcTerminals210_2BK1250.A_0010_KL_6211_ASI_Master_Parameter_Interface_and_32_Byte_62_ASI_Slaves_Power.Channel_1.ASI_Out_Slave_2 <-> Channel 1/ASI Out Slave 2
//     PlcTask Outputs/GVL_iXlinker.EtherCAT_Master_BKCUCX.TcTerminals210_EK1100_2.TcTerminals210_2BK1250.A_0010_KL_6211_ASI_Master_Parameter_Interface_and_32_Byte_62_ASI_Slaves_Power.Channel_1.ASI_Out_Slave_3 <-> Channel 1/ASI Out Slave 3
//     PlcTask Outputs/GVL_iXlinker.EtherCAT_Master_BKCUCX.TcTerminals210_EK1100_2.TcTerminals210_2BK1250.A_0010_KL_6211_ASI_Master_Parameter_Interface_and_32_Byte_62_ASI_Slaves_Power.Channel_1.ASI_Out_Slave_4 <-> Channel 1/ASI Out Slave 4
//     PlcTask Outputs/GVL_iXlinker.EtherCAT_Master_BKCUCX.TcTerminals210_EK1100_2.TcTerminals210_2BK1250.A_0010_KL_6211_ASI_Master_Parameter_Interface_and_32_Byte_62_ASI_Slaves_Power.Channel_1.ASI_Out_Slave_5 <-> Channel 1/ASI Out Slave 5
//     PlcTask Outputs/GVL_iXlinker.EtherCAT_Master_BKCUCX.TcTerminals210_EK1100_2.TcTerminals210_2BK1250.A_0010_KL_6211_ASI_Master_Parameter_Interface_and_32_Byte_62_ASI_Slaves_Power.Channel_1.ASI_Out_Slave_6 <-> Channel 1/ASI Out Slave 6
//     PlcTask Outputs/GVL_iXlinker.EtherCAT_Master_BKCUCX.TcTerminals210_EK1100_2.TcTerminals210_2BK1250.A_0010_KL_6211_ASI_Master_Parameter_Interface_and_32_Byte_62_ASI_Slaves_Power.Channel_1.ASI_Out_Slave_7 <-> Channel 1/ASI Out Slave 7
//     PlcTask Outputs/GVL_iXlinker.EtherCAT_Master_BKCUCX.TcTerminals210_EK1100_2.TcTerminals210_2BK1250.A_0010_KL_6211_ASI_Master_Parameter_Interface_and_32_Byte_62_ASI_Slaves_Power.Channel_1.ASI_Out_Slave_8 <-> Channel 1/ASI Out Slave 8
//     PlcTask Outputs/GVL_iXlinker.EtherCAT_Master_BKCUCX.TcTerminals210_EK1100_2.TcTerminals210_2BK1250.A_0010_KL_6211_ASI_Master_Parameter_Interface_and_32_Byte_62_ASI_Slaves_Power.Channel_1.ASI_Out_Slave_9 <-> Channel 1/ASI Out Slave 9
//     PlcTask Outputs/GVL_iXlinker.EtherCAT_Master_BKCUCX.TcTerminals210_EK1100_2.TcTerminals210_2BK1250.A_0010_KL_6211_ASI_Master_Parameter_Interface_and_32_Byte_62_ASI_Slaves_Power.Channel_1.ASI_Out_Slave_10 <-> Channel 1/ASI Out Slave 10
//     PlcTask Outputs/GVL_iXlinker.EtherCAT_Master_BKCUCX.TcTerminals210_EK1100_2.TcTerminals210_2BK1250.A_0010_KL_6211_ASI_Master_Parameter_Interface_and_32_Byte_62_ASI_Slaves_Power.Channel_1.ASI_Out_Slave_11 <-> Channel 1/ASI Out Slave 11
//     PlcTask Outputs/GVL_iXlinker.EtherCAT_Master_BKCUCX.TcTerminals210_EK1100_2.TcTerminals210_2BK1250.A_0010_KL_6211_ASI_Master_Parameter_Interface_and_32_Byte_62_ASI_Slaves_Power.Channel_1.ASI_Out_Slave_12 <-> Channel 1/ASI Out Slave 12
//     PlcTask Outputs/GVL_iXlinker.EtherCAT_Master_BKCUCX.TcTerminals210_EK1100_2.TcTerminals210_2BK1250.A_0010_KL_6211_ASI_Master_Parameter_Interface_and_32_Byte_62_ASI_Slaves_Power.Channel_1.ASI_Out_Slave_13 <-> Channel 1/ASI Out Slave 13
//     PlcTask Outputs/GVL_iXlinker.EtherCAT_Master_BKCUCX.TcTerminals210_EK1100_2.TcTerminals210_2BK1250.A_0010_KL_6211_ASI_Master_Parameter_Interface_and_32_Byte_62_ASI_Slaves_Power.Channel_1.ASI_Out_Slave_14 <-> Channel 1/ASI Out Slave 14
//     PlcTask Outputs/GVL_iXlinker.EtherCAT_Master_BKCUCX.TcTerminals210_EK1100_2.TcTerminals210_2BK1250.A_0010_KL_6211_ASI_Master_Parameter_Interface_and_32_Byte_62_ASI_Slaves_Power.Channel_1.ASI_Out_Slave_15 <-> Channel 1/ASI Out Slave 15
//     PlcTask Outputs/GVL_iXlinker.EtherCAT_Master_BKCUCX.TcTerminals210_EK1100_2.TcTerminals210_2BK1250.A_0010_KL_6211_ASI_Master_Parameter_Interface_and_32_Byte_62_ASI_Slaves_Power.Channel_1.ASI_Out_Slave_16 <-> Channel 1/ASI Out Slave 16
//     PlcTask Outputs/GVL_iXlinker.EtherCAT_Master_BKCUCX.TcTerminals210_EK1100_2.TcTerminals210_2BK1250.A_0010_KL_6211_ASI_Master_Parameter_Interface_and_32_Byte_62_ASI_Slaves_Power.Channel_1.ASI_Out_Slave_17 <-> Channel 1/ASI Out Slave 17
//     PlcTask Outputs/GVL_iXlinker.EtherCAT_Master_BKCUCX.TcTerminals210_EK1100_2.TcTerminals210_2BK1250.A_0010_KL_6211_ASI_Master_Parameter_Interface_and_32_Byte_62_ASI_Slaves_Power.Channel_1.ASI_Out_Slave_18 <-> Channel 1/ASI Out Slave 18
//     PlcTask Outputs/GVL_iXlinker.EtherCAT_Master_BKCUCX.TcTerminals210_EK1100_2.TcTerminals210_2BK1250.A_0010_KL_6211_ASI_Master_Parameter_Interface_and_32_Byte_62_ASI_Slaves_Power.Channel_1.ASI_Out_Slave_19 <-> Channel 1/ASI Out Slave 19
//     PlcTask Outputs/GVL_iXlinker.EtherCAT_Master_BKCUCX.TcTerminals210_EK1100_2.TcTerminals210_2BK1250.A_0010_KL_6211_ASI_Master_Parameter_Interface_and_32_Byte_62_ASI_Slaves_Power.Channel_1.ASI_Out_Slave_20 <-> Channel 1/ASI Out Slave 20
//     PlcTask Outputs/GVL_iXlinker.EtherCAT_Master_BKCUCX.TcTerminals210_EK1100_2.TcTerminals210_2BK1250.A_0010_KL_6211_ASI_Master_Parameter_Interface_and_32_Byte_62_ASI_Slaves_Power.Channel_1.ASI_Out_Slave_21 <-> Channel 1/ASI Out Slave 21
//     PlcTask Outputs/GVL_iXlinker.EtherCAT_Master_BKCUCX.TcTerminals210_EK1100_2.TcTerminals210_2BK1250.A_0010_KL_6211_ASI_Master_Parameter_Interface_and_32_Byte_62_ASI_Slaves_Power.Channel_1.ASI_Out_Slave_22 <-> Channel 1/ASI Out Slave 22
//     PlcTask Outputs/GVL_iXlinker.EtherCAT_Master_BKCUCX.TcTerminals210_EK1100_2.TcTerminals210_2BK1250.A_0010_KL_6211_ASI_Master_Parameter_Interface_and_32_Byte_62_ASI_Slaves_Power.Channel_1.ASI_Out_Slave_23 <-> Channel 1/ASI Out Slave 23
//     PlcTask Outputs/GVL_iXlinker.EtherCAT_Master_BKCUCX.TcTerminals210_EK1100_2.TcTerminals210_2BK1250.A_0010_KL_6211_ASI_Master_Parameter_Interface_and_32_Byte_62_ASI_Slaves_Power.Channel_1.ASI_Out_Slave_24 <-> Channel 1/ASI Out Slave 24
//     PlcTask Outputs/GVL_iXlinker.EtherCAT_Master_BKCUCX.TcTerminals210_EK1100_2.TcTerminals210_2BK1250.A_0010_KL_6211_ASI_Master_Parameter_Interface_and_32_Byte_62_ASI_Slaves_Power.Channel_1.ASI_Out_Slave_25 <-> Channel 1/ASI Out Slave 25
//     PlcTask Outputs/GVL_iXlinker.EtherCAT_Master_BKCUCX.TcTerminals210_EK1100_2.TcTerminals210_2BK1250.A_0010_KL_6211_ASI_Master_Parameter_Interface_and_32_Byte_62_ASI_Slaves_Power.Channel_1.ASI_Out_Slave_26 <-> Channel 1/ASI Out Slave 26
//     PlcTask Outputs/GVL_iXlinker.EtherCAT_Master_BKCUCX.TcTerminals210_EK1100_2.TcTerminals210_2BK1250.A_0010_KL_6211_ASI_Master_Parameter_Interface_and_32_Byte_62_ASI_Slaves_Power.Channel_1.ASI_Out_Slave_27 <-> Channel 1/ASI Out Slave 27
//     PlcTask Outputs/GVL_iXlinker.EtherCAT_Master_BKCUCX.TcTerminals210_EK1100_2.TcTerminals210_2BK1250.A_0010_KL_6211_ASI_Master_Parameter_Interface_and_32_Byte_62_ASI_Slaves_Power.Channel_1.ASI_Out_Slave_28 <-> Channel 1/ASI Out Slave 28
//     PlcTask Outputs/GVL_iXlinker.EtherCAT_Master_BKCUCX.TcTerminals210_EK1100_2.TcTerminals210_2BK1250.A_0010_KL_6211_ASI_Master_Parameter_Interface_and_32_Byte_62_ASI_Slaves_Power.Channel_1.ASI_Out_Slave_29 <-> Channel 1/ASI Out Slave 29
//     PlcTask Outputs/GVL_iXlinker.EtherCAT_Master_BKCUCX.TcTerminals210_EK1100_2.TcTerminals210_2BK1250.A_0010_KL_6211_ASI_Master_Parameter_Interface_and_32_Byte_62_ASI_Slaves_Power.Channel_1.ASI_Out_Slave_30 <-> Channel 1/ASI Out Slave 30
//     PlcTask Outputs/GVL_iXlinker.EtherCAT_Master_BKCUCX.TcTerminals210_EK1100_2.TcTerminals210_2BK1250.A_0010_KL_6211_ASI_Master_Parameter_Interface_and_32_Byte_62_ASI_Slaves_Power.Channel_1.ASI_Out_Slave_31 <-> Channel 1/ASI Out Slave 31
//     PlcTask Outputs/GVL_iXlinker.EtherCAT_Master_BKCUCX.TcTerminals210_EK1100_2.TcTerminals210_2BK1250.A_0010_KL_6211_ASI_Master_Parameter_Interface_and_32_Byte_62_ASI_Slaves_Power.Channel_1.ASI_Out_Slave_32 <-> Channel 1/ASI Out Slave 32
//     PlcTask Outputs/GVL_iXlinker.EtherCAT_Master_BKCUCX.TcTerminals210_EK1100_2.TcTerminals210_2BK1250.A_0010_KL_6211_ASI_Master_Parameter_Interface_and_32_Byte_62_ASI_Slaves_Power.Channel_1.ASI_Out_Slave_33 <-> Channel 1/ASI Out Slave 33
//     PlcTask Outputs/GVL_iXlinker.EtherCAT_Master_BKCUCX.TcTerminals210_EK1100_2.TcTerminals210_2BK1250.A_0010_KL_6211_ASI_Master_Parameter_Interface_and_32_Byte_62_ASI_Slaves_Power.Channel_1.ASI_Out_Slave_34 <-> Channel 1/ASI Out Slave 34
//     PlcTask Outputs/GVL_iXlinker.EtherCAT_Master_BKCUCX.TcTerminals210_EK1100_2.TcTerminals210_2BK1250.A_0010_KL_6211_ASI_Master_Parameter_Interface_and_32_Byte_62_ASI_Slaves_Power.Channel_1.ASI_Out_Slave_35 <-> Channel 1/ASI Out Slave 35
//     PlcTask Outputs/GVL_iXlinker.EtherCAT_Master_BKCUCX.TcTerminals210_EK1100_2.TcTerminals210_2BK1250.A_0010_KL_6211_ASI_Master_Parameter_Interface_and_32_Byte_62_ASI_Slaves_Power.Channel_1.ASI_Out_Slave_36 <-> Channel 1/ASI Out Slave 36
//     PlcTask Outputs/GVL_iXlinker.EtherCAT_Master_BKCUCX.TcTerminals210_EK1100_2.TcTerminals210_2BK1250.A_0010_KL_6211_ASI_Master_Parameter_Interface_and_32_Byte_62_ASI_Slaves_Power.Channel_1.ASI_Out_Slave_37 <-> Channel 1/ASI Out Slave 37
//     PlcTask Outputs/GVL_iXlinker.EtherCAT_Master_BKCUCX.TcTerminals210_EK1100_2.TcTerminals210_2BK1250.A_0010_KL_6211_ASI_Master_Parameter_Interface_and_32_Byte_62_ASI_Slaves_Power.Channel_1.ASI_Out_Slave_38 <-> Channel 1/ASI Out Slave 38
//     PlcTask Outputs/GVL_iXlinker.EtherCAT_Master_BKCUCX.TcTerminals210_EK1100_2.TcTerminals210_2BK1250.A_0010_KL_6211_ASI_Master_Parameter_Interface_and_32_Byte_62_ASI_Slaves_Power.Channel_1.ASI_Out_Slave_39 <-> Channel 1/ASI Out Slave 39
//     PlcTask Outputs/GVL_iXlinker.EtherCAT_Master_BKCUCX.TcTerminals210_EK1100_2.TcTerminals210_2BK1250.A_0010_KL_6211_ASI_Master_Parameter_Interface_and_32_Byte_62_ASI_Slaves_Power.Channel_1.ASI_Out_Slave_40 <-> Channel 1/ASI Out Slave 40
//     PlcTask Outputs/GVL_iXlinker.EtherCAT_Master_BKCUCX.TcTerminals210_EK1100_2.TcTerminals210_2BK1250.A_0010_KL_6211_ASI_Master_Parameter_Interface_and_32_Byte_62_ASI_Slaves_Power.Channel_1.ASI_Out_Slave_41 <-> Channel 1/ASI Out Slave 41
//     PlcTask Outputs/GVL_iXlinker.EtherCAT_Master_BKCUCX.TcTerminals210_EK1100_2.TcTerminals210_2BK1250.A_0010_KL_6211_ASI_Master_Parameter_Interface_and_32_Byte_62_ASI_Slaves_Power.Channel_1.ASI_Out_Slave_42 <-> Channel 1/ASI Out Slave 42
//     PlcTask Outputs/GVL_iXlinker.EtherCAT_Master_BKCUCX.TcTerminals210_EK1100_2.TcTerminals210_2BK1250.A_0010_KL_6211_ASI_Master_Parameter_Interface_and_32_Byte_62_ASI_Slaves_Power.Channel_1.ASI_Out_Slave_43 <-> Channel 1/ASI Out Slave 43
//     PlcTask Outputs/GVL_iXlinker.EtherCAT_Master_BKCUCX.TcTerminals210_EK1100_2.TcTerminals210_2BK1250.A_0010_KL_6211_ASI_Master_Parameter_Interface_and_32_Byte_62_ASI_Slaves_Power.Channel_1.ASI_Out_Slave_44 <-> Channel 1/ASI Out Slave 44
//     PlcTask Outputs/GVL_iXlinker.EtherCAT_Master_BKCUCX.TcTerminals210_EK1100_2.TcTerminals210_2BK1250.A_0010_KL_6211_ASI_Master_Parameter_Interface_and_32_Byte_62_ASI_Slaves_Power.Channel_1.ASI_Out_Slave_45 <-> Channel 1/ASI Out Slave 45
//     PlcTask Outputs/GVL_iXlinker.EtherCAT_Master_BKCUCX.TcTerminals210_EK1100_2.TcTerminals210_2BK1250.A_0010_KL_6211_ASI_Master_Parameter_Interface_and_32_Byte_62_ASI_Slaves_Power.Channel_1.ASI_Out_Slave_46 <-> Channel 1/ASI Out Slave 46
//     PlcTask Outputs/GVL_iXlinker.EtherCAT_Master_BKCUCX.TcTerminals210_EK1100_2.TcTerminals210_2BK1250.A_0010_KL_6211_ASI_Master_Parameter_Interface_and_32_Byte_62_ASI_Slaves_Power.Channel_1.ASI_Out_Slave_47 <-> Channel 1/ASI Out Slave 47
//     PlcTask Outputs/GVL_iXlinker.EtherCAT_Master_BKCUCX.TcTerminals210_EK1100_2.TcTerminals210_2BK1250.A_0010_KL_6211_ASI_Master_Parameter_Interface_and_32_Byte_62_ASI_Slaves_Power.Channel_1.ASI_Out_Slave_48 <-> Channel 1/ASI Out Slave 48
//     PlcTask Outputs/GVL_iXlinker.EtherCAT_Master_BKCUCX.TcTerminals210_EK1100_2.TcTerminals210_2BK1250.A_0010_KL_6211_ASI_Master_Parameter_Interface_and_32_Byte_62_ASI_Slaves_Power.Channel_1.ASI_Out_Slave_49 <-> Channel 1/ASI Out Slave 49
//     PlcTask Outputs/GVL_iXlinker.EtherCAT_Master_BKCUCX.TcTerminals210_EK1100_2.TcTerminals210_2BK1250.A_0010_KL_6211_ASI_Master_Parameter_Interface_and_32_Byte_62_ASI_Slaves_Power.Channel_1.ASI_Out_Slave_50 <-> Channel 1/ASI Out Slave 50
//     PlcTask Outputs/GVL_iXlinker.EtherCAT_Master_BKCUCX.TcTerminals210_EK1100_2.TcTerminals210_2BK1250.A_0010_KL_6211_ASI_Master_Parameter_Interface_and_32_Byte_62_ASI_Slaves_Power.Channel_1.ASI_Out_Slave_51 <-> Channel 1/ASI Out Slave 51
//     PlcTask Outputs/GVL_iXlinker.EtherCAT_Master_BKCUCX.TcTerminals210_EK1100_2.TcTerminals210_2BK1250.A_0010_KL_6211_ASI_Master_Parameter_Interface_and_32_Byte_62_ASI_Slaves_Power.Channel_1.ASI_Out_Slave_52 <-> Channel 1/ASI Out Slave 52
//     PlcTask Outputs/GVL_iXlinker.EtherCAT_Master_BKCUCX.TcTerminals210_EK1100_2.TcTerminals210_2BK1250.A_0010_KL_6211_ASI_Master_Parameter_Interface_and_32_Byte_62_ASI_Slaves_Power.Channel_1.ASI_Out_Slave_53 <-> Channel 1/ASI Out Slave 53
//     PlcTask Outputs/GVL_iXlinker.EtherCAT_Master_BKCUCX.TcTerminals210_EK1100_2.TcTerminals210_2BK1250.A_0010_KL_6211_ASI_Master_Parameter_Interface_and_32_Byte_62_ASI_Slaves_Power.Channel_1.ASI_Out_Slave_54 <-> Channel 1/ASI Out Slave 54
//     PlcTask Outputs/GVL_iXlinker.EtherCAT_Master_BKCUCX.TcTerminals210_EK1100_2.TcTerminals210_2BK1250.A_0010_KL_6211_ASI_Master_Parameter_Interface_and_32_Byte_62_ASI_Slaves_Power.Channel_1.ASI_Out_Slave_55 <-> Channel 1/ASI Out Slave 55
//     PlcTask Outputs/GVL_iXlinker.EtherCAT_Master_BKCUCX.TcTerminals210_EK1100_2.TcTerminals210_2BK1250.A_0010_KL_6211_ASI_Master_Parameter_Interface_and_32_Byte_62_ASI_Slaves_Power.Channel_1.ASI_Out_Slave_56 <-> Channel 1/ASI Out Slave 56
//     PlcTask Outputs/GVL_iXlinker.EtherCAT_Master_BKCUCX.TcTerminals210_EK1100_2.TcTerminals210_2BK1250.A_0010_KL_6211_ASI_Master_Parameter_Interface_and_32_Byte_62_ASI_Slaves_Power.Channel_1.ASI_Out_Slave_57 <-> Channel 1/ASI Out Slave 57
//     PlcTask Outputs/GVL_iXlinker.EtherCAT_Master_BKCUCX.TcTerminals210_EK1100_2.TcTerminals210_2BK1250.A_0010_KL_6211_ASI_Master_Parameter_Interface_and_32_Byte_62_ASI_Slaves_Power.Channel_1.ASI_Out_Slave_58 <-> Channel 1/ASI Out Slave 58
//     PlcTask Outputs/GVL_iXlinker.EtherCAT_Master_BKCUCX.TcTerminals210_EK1100_2.TcTerminals210_2BK1250.A_0010_KL_6211_ASI_Master_Parameter_Interface_and_32_Byte_62_ASI_Slaves_Power.Channel_1.ASI_Out_Slave_59 <-> Channel 1/ASI Out Slave 59
//     PlcTask Outputs/GVL_iXlinker.EtherCAT_Master_BKCUCX.TcTerminals210_EK1100_2.TcTerminals210_2BK1250.A_0010_KL_6211_ASI_Master_Parameter_Interface_and_32_Byte_62_ASI_Slaves_Power.Channel_1.ASI_Out_Slave_60 <-> Channel 1/ASI Out Slave 60
//     PlcTask Outputs/GVL_iXlinker.EtherCAT_Master_BKCUCX.TcTerminals210_EK1100_2.TcTerminals210_2BK1250.A_0010_KL_6211_ASI_Master_Parameter_Interface_and_32_Byte_62_ASI_Slaves_Power.Channel_1.ASI_Out_Slave_61 <-> Channel 1/ASI Out Slave 61
//     PlcTask Outputs/GVL_iXlinker.EtherCAT_Master_BKCUCX.TcTerminals210_EK1100_2.TcTerminals210_2BK1250.A_0010_KL_6211_ASI_Master_Parameter_Interface_and_32_Byte_62_ASI_Slaves_Power.Channel_1.ASI_Out_Slave_62 <-> Channel 1/ASI Out Slave 62
//     PlcTask Outputs/GVL_iXlinker.EtherCAT_Master_BKCUCX.TcTerminals210_EK1100_2.TcTerminals210_2BK1250.A_0010_KL_6211_ASI_Master_Parameter_Interface_and_32_Byte_62_ASI_Slaves_Power.Channel_1.ASI_Out_Slave_63 <-> Channel 1/ASI Out Slave 63
//   PLC/PLC Instance <-> EtherCAT Master BKCUCX/TcTerminals210_EK1100_2/TcTerminals210_2BK1250/A_0012(KL 6224 IO-Link-Master (Parameter Interface and 6 Byte Process Data)
//     PlcTask Inputs/GVL_iXlinker.EtherCAT_Master_BKCUCX.TcTerminals210_EK1100_2.TcTerminals210_2BK1250.A_0012_KL_6224_IO_Link_Master_Parameter_Interface_and_6_Byte_Process_Data.Channel_1.Status <-> Channel 1/Status
//     PlcTask Inputs/GVL_iXlinker.EtherCAT_Master_BKCUCX.TcTerminals210_EK1100_2.TcTerminals210_2BK1250.A_0012_KL_6224_IO_Link_Master_Parameter_Interface_and_6_Byte_Process_Data.Channel_1.Parameter_In <-> Channel 1/Parameter In
//     PlcTask Inputs/GVL_iXlinker.EtherCAT_Master_BKCUCX.TcTerminals210_EK1100_2.TcTerminals210_2BK1250.A_0012_KL_6224_IO_Link_Master_Parameter_Interface_and_6_Byte_Process_Data.Channel_1.State_Ch1 <-> Channel 1/State Ch1
//     PlcTask Inputs/GVL_iXlinker.EtherCAT_Master_BKCUCX.TcTerminals210_EK1100_2.TcTerminals210_2BK1250.A_0012_KL_6224_IO_Link_Master_Parameter_Interface_and_6_Byte_Process_Data.Channel_1.State_Ch2 <-> Channel 1/State Ch2
//     PlcTask Inputs/GVL_iXlinker.EtherCAT_Master_BKCUCX.TcTerminals210_EK1100_2.TcTerminals210_2BK1250.A_0012_KL_6224_IO_Link_Master_Parameter_Interface_and_6_Byte_Process_Data.Channel_1.State_Ch3 <-> Channel 1/State Ch3
//     PlcTask Inputs/GVL_iXlinker.EtherCAT_Master_BKCUCX.TcTerminals210_EK1100_2.TcTerminals210_2BK1250.A_0012_KL_6224_IO_Link_Master_Parameter_Interface_and_6_Byte_Process_Data.Channel_1.State_Ch4 <-> Channel 1/State Ch4
//     PlcTask Inputs/GVL_iXlinker.EtherCAT_Master_BKCUCX.TcTerminals210_EK1100_2.TcTerminals210_2BK1250.A_0012_KL_6224_IO_Link_Master_Parameter_Interface_and_6_Byte_Process_Data.Channel_1.Data_In_0 <-> Channel 1/Data In 0
//     PlcTask Inputs/GVL_iXlinker.EtherCAT_Master_BKCUCX.TcTerminals210_EK1100_2.TcTerminals210_2BK1250.A_0012_KL_6224_IO_Link_Master_Parameter_Interface_and_6_Byte_Process_Data.Channel_1.Data_In_1 <-> Channel 1/Data In 1
//     PlcTask Outputs/GVL_iXlinker.EtherCAT_Master_BKCUCX.TcTerminals210_EK1100_2.TcTerminals210_2BK1250.A_0012_KL_6224_IO_Link_Master_Parameter_Interface_and_6_Byte_Process_Data.Channel_1.Control <-> Channel 1/Control
//     PlcTask Outputs/GVL_iXlinker.EtherCAT_Master_BKCUCX.TcTerminals210_EK1100_2.TcTerminals210_2BK1250.A_0012_KL_6224_IO_Link_Master_Parameter_Interface_and_6_Byte_Process_Data.Channel_1.Parameter_Out <-> Channel 1/Parameter Out
//     PlcTask Outputs/GVL_iXlinker.EtherCAT_Master_BKCUCX.TcTerminals210_EK1100_2.TcTerminals210_2BK1250.A_0012_KL_6224_IO_Link_Master_Parameter_Interface_and_6_Byte_Process_Data.Channel_1.Data_Out_0 <-> Channel 1/Data Out 0
//     PlcTask Outputs/GVL_iXlinker.EtherCAT_Master_BKCUCX.TcTerminals210_EK1100_2.TcTerminals210_2BK1250.A_0012_KL_6224_IO_Link_Master_Parameter_Interface_and_6_Byte_Process_Data.Channel_1.Data_Out_1 <-> Channel 1/Data Out 1
//     PlcTask Outputs/GVL_iXlinker.EtherCAT_Master_BKCUCX.TcTerminals210_EK1100_2.TcTerminals210_2BK1250.A_0012_KL_6224_IO_Link_Master_Parameter_Interface_and_6_Byte_Process_Data.Channel_1.Data_Out_2 <-> Channel 1/Data Out 2
//     PlcTask Outputs/GVL_iXlinker.EtherCAT_Master_BKCUCX.TcTerminals210_EK1100_2.TcTerminals210_2BK1250.A_0012_KL_6224_IO_Link_Master_Parameter_Interface_and_6_Byte_Process_Data.Channel_1.Data_Out_3 <-> Channel 1/Data Out 3
//     PlcTask Outputs/GVL_iXlinker.EtherCAT_Master_BKCUCX.TcTerminals210_EK1100_2.TcTerminals210_2BK1250.A_0012_KL_6224_IO_Link_Master_Parameter_Interface_and_6_Byte_Process_Data.Channel_1.Data_Out_4 <-> Channel 1/Data Out 4
//     PlcTask Outputs/GVL_iXlinker.EtherCAT_Master_BKCUCX.TcTerminals210_EK1100_2.TcTerminals210_2BK1250.A_0012_KL_6224_IO_Link_Master_Parameter_Interface_and_6_Byte_Process_Data.Channel_1.Data_Out_5 <-> Channel 1/Data Out 5
//   PLC/PLC Instance <-> EtherCAT Master BKCUCX/TcTerminals210_EK1100_2/TcTerminals210_2BK1250/A_0013(KL 6224 IO-Link-Master (Parameter Interface and 18 Byte Process Data)
//     PlcTask Inputs/GVL_iXlinker.EtherCAT_Master_BKCUCX.TcTerminals210_EK1100_2.TcTerminals210_2BK1250.A_0013_KL_6224_IO_Link_Master_Parameter_Interface_and_18_Byte_Process_Data.Channel_1.Status <-> Channel 1/Status
//     PlcTask Inputs/GVL_iXlinker.EtherCAT_Master_BKCUCX.TcTerminals210_EK1100_2.TcTerminals210_2BK1250.A_0013_KL_6224_IO_Link_Master_Parameter_Interface_and_18_Byte_Process_Data.Channel_1.Parameter_In <-> Channel 1/Parameter In
//     PlcTask Inputs/GVL_iXlinker.EtherCAT_Master_BKCUCX.TcTerminals210_EK1100_2.TcTerminals210_2BK1250.A_0013_KL_6224_IO_Link_Master_Parameter_Interface_and_18_Byte_Process_Data.Channel_1.State_Ch1 <-> Channel 1/State Ch1
//     PlcTask Inputs/GVL_iXlinker.EtherCAT_Master_BKCUCX.TcTerminals210_EK1100_2.TcTerminals210_2BK1250.A_0013_KL_6224_IO_Link_Master_Parameter_Interface_and_18_Byte_Process_Data.Channel_1.State_Ch2 <-> Channel 1/State Ch2
//     PlcTask Inputs/GVL_iXlinker.EtherCAT_Master_BKCUCX.TcTerminals210_EK1100_2.TcTerminals210_2BK1250.A_0013_KL_6224_IO_Link_Master_Parameter_Interface_and_18_Byte_Process_Data.Channel_1.State_Ch3 <-> Channel 1/State Ch3
//     PlcTask Inputs/GVL_iXlinker.EtherCAT_Master_BKCUCX.TcTerminals210_EK1100_2.TcTerminals210_2BK1250.A_0013_KL_6224_IO_Link_Master_Parameter_Interface_and_18_Byte_Process_Data.Channel_1.State_Ch4 <-> Channel 1/State Ch4
//     PlcTask Inputs/GVL_iXlinker.EtherCAT_Master_BKCUCX.TcTerminals210_EK1100_2.TcTerminals210_2BK1250.A_0013_KL_6224_IO_Link_Master_Parameter_Interface_and_18_Byte_Process_Data.Channel_1.Data_In_0 <-> Channel 1/Data In 0
//     PlcTask Inputs/GVL_iXlinker.EtherCAT_Master_BKCUCX.TcTerminals210_EK1100_2.TcTerminals210_2BK1250.A_0013_KL_6224_IO_Link_Master_Parameter_Interface_and_18_Byte_Process_Data.Channel_1.Data_In_1 <-> Channel 1/Data In 1
//     PlcTask Inputs/GVL_iXlinker.EtherCAT_Master_BKCUCX.TcTerminals210_EK1100_2.TcTerminals210_2BK1250.A_0013_KL_6224_IO_Link_Master_Parameter_Interface_and_18_Byte_Process_Data.Channel_1.Data_In_2 <-> Channel 1/Data In 2
//     PlcTask Inputs/GVL_iXlinker.EtherCAT_Master_BKCUCX.TcTerminals210_EK1100_2.TcTerminals210_2BK1250.A_0013_KL_6224_IO_Link_Master_Parameter_Interface_and_18_Byte_Process_Data.Channel_1.Data_In_3 <-> Channel 1/Data In 3
//     PlcTask Inputs/GVL_iXlinker.EtherCAT_Master_BKCUCX.TcTerminals210_EK1100_2.TcTerminals210_2BK1250.A_0013_KL_6224_IO_Link_Master_Parameter_Interface_and_18_Byte_Process_Data.Channel_1.Data_In_4 <-> Channel 1/Data In 4
//     PlcTask Inputs/GVL_iXlinker.EtherCAT_Master_BKCUCX.TcTerminals210_EK1100_2.TcTerminals210_2BK1250.A_0013_KL_6224_IO_Link_Master_Parameter_Interface_and_18_Byte_Process_Data.Channel_1.Data_In_5 <-> Channel 1/Data In 5
//     PlcTask Inputs/GVL_iXlinker.EtherCAT_Master_BKCUCX.TcTerminals210_EK1100_2.TcTerminals210_2BK1250.A_0013_KL_6224_IO_Link_Master_Parameter_Interface_and_18_Byte_Process_Data.Channel_1.Data_In_6 <-> Channel 1/Data In 6
//     PlcTask Inputs/GVL_iXlinker.EtherCAT_Master_BKCUCX.TcTerminals210_EK1100_2.TcTerminals210_2BK1250.A_0013_KL_6224_IO_Link_Master_Parameter_Interface_and_18_Byte_Process_Data.Channel_1.Data_In_7 <-> Channel 1/Data In 7
//     PlcTask Inputs/GVL_iXlinker.EtherCAT_Master_BKCUCX.TcTerminals210_EK1100_2.TcTerminals210_2BK1250.A_0013_KL_6224_IO_Link_Master_Parameter_Interface_and_18_Byte_Process_Data.Channel_1.Data_In_8 <-> Channel 1/Data In 8
//     PlcTask Inputs/GVL_iXlinker.EtherCAT_Master_BKCUCX.TcTerminals210_EK1100_2.TcTerminals210_2BK1250.A_0013_KL_6224_IO_Link_Master_Parameter_Interface_and_18_Byte_Process_Data.Channel_1.Data_In_9 <-> Channel 1/Data In 9
//     PlcTask Inputs/GVL_iXlinker.EtherCAT_Master_BKCUCX.TcTerminals210_EK1100_2.TcTerminals210_2BK1250.A_0013_KL_6224_IO_Link_Master_Parameter_Interface_and_18_Byte_Process_Data.Channel_1.Data_In_10 <-> Channel 1/Data In 10
//     PlcTask Inputs/GVL_iXlinker.EtherCAT_Master_BKCUCX.TcTerminals210_EK1100_2.TcTerminals210_2BK1250.A_0013_KL_6224_IO_Link_Master_Parameter_Interface_and_18_Byte_Process_Data.Channel_1.Data_In_11 <-> Channel 1/Data In 11
//     PlcTask Inputs/GVL_iXlinker.EtherCAT_Master_BKCUCX.TcTerminals210_EK1100_2.TcTerminals210_2BK1250.A_0013_KL_6224_IO_Link_Master_Parameter_Interface_and_18_Byte_Process_Data.Channel_1.Data_In_12 <-> Channel 1/Data In 12
//     PlcTask Inputs/GVL_iXlinker.EtherCAT_Master_BKCUCX.TcTerminals210_EK1100_2.TcTerminals210_2BK1250.A_0013_KL_6224_IO_Link_Master_Parameter_Interface_and_18_Byte_Process_Data.Channel_1.Data_In_13 <-> Channel 1/Data In 13
//     PlcTask Outputs/GVL_iXlinker.EtherCAT_Master_BKCUCX.TcTerminals210_EK1100_2.TcTerminals210_2BK1250.A_0013_KL_6224_IO_Link_Master_Parameter_Interface_and_18_Byte_Process_Data.Channel_1.Control <-> Channel 1/Control
//     PlcTask Outputs/GVL_iXlinker.EtherCAT_Master_BKCUCX.TcTerminals210_EK1100_2.TcTerminals210_2BK1250.A_0013_KL_6224_IO_Link_Master_Parameter_Interface_and_18_Byte_Process_Data.Channel_1.Parameter_Out <-> Channel 1/Parameter Out
//     PlcTask Outputs/GVL_iXlinker.EtherCAT_Master_BKCUCX.TcTerminals210_EK1100_2.TcTerminals210_2BK1250.A_0013_KL_6224_IO_Link_Master_Parameter_Interface_and_18_Byte_Process_Data.Channel_1.Data_Out_0 <-> Channel 1/Data Out 0
//     PlcTask Outputs/GVL_iXlinker.EtherCAT_Master_BKCUCX.TcTerminals210_EK1100_2.TcTerminals210_2BK1250.A_0013_KL_6224_IO_Link_Master_Parameter_Interface_and_18_Byte_Process_Data.Channel_1.Data_Out_1 <-> Channel 1/Data Out 1
//     PlcTask Outputs/GVL_iXlinker.EtherCAT_Master_BKCUCX.TcTerminals210_EK1100_2.TcTerminals210_2BK1250.A_0013_KL_6224_IO_Link_Master_Parameter_Interface_and_18_Byte_Process_Data.Channel_1.Data_Out_2 <-> Channel 1/Data Out 2
//     PlcTask Outputs/GVL_iXlinker.EtherCAT_Master_BKCUCX.TcTerminals210_EK1100_2.TcTerminals210_2BK1250.A_0013_KL_6224_IO_Link_Master_Parameter_Interface_and_18_Byte_Process_Data.Channel_1.Data_Out_3 <-> Channel 1/Data Out 3
//     PlcTask Outputs/GVL_iXlinker.EtherCAT_Master_BKCUCX.TcTerminals210_EK1100_2.TcTerminals210_2BK1250.A_0013_KL_6224_IO_Link_Master_Parameter_Interface_and_18_Byte_Process_Data.Channel_1.Data_Out_4 <-> Channel 1/Data Out 4
//     PlcTask Outputs/GVL_iXlinker.EtherCAT_Master_BKCUCX.TcTerminals210_EK1100_2.TcTerminals210_2BK1250.A_0013_KL_6224_IO_Link_Master_Parameter_Interface_and_18_Byte_Process_Data.Channel_1.Data_Out_5 <-> Channel 1/Data Out 5
